(* IEC 61131-3 sources: volt/packages/volt-lsp-iec/test-corpus/lenze-mid/Device/Plc Logic/Application/Library Manager/L_MC4P_RoboticHandling (part 3) *)

(* ---- L_MC4P_KIN_REF_GENERIC.pou ---- *)
FUNCTION_BLOCK L_MC4P_KIN_REF_GENERIC
VAR_OUTPUT
	XACTIVE : BOOL;
END_VAR
VAR
	PAXESGROUP : POINTER TO Axes_Group_KIN;
END_VAR
END_FUNCTION_BLOCK

METHOD GETPARAITF : L_MC4P_IKinParamExtern
END_METHOD

METHOD GETTRAFOITF : L_MC4P_ITrafoExtern
END_METHOD

METHOD LINKEDAXESGROUP_GET : POINTER TO AXES_GROUP_KIN
END_METHOD

METHOD LINKEDAXESGROUP_SET
VAR_INPUT
	LINKEDAXESGROUP : POINTER TO AXES_GROUP_KIN;
END_VAR
END_METHOD

METHOD SETACSAXISTYPE
VAR_OUTPUT
	AEAXES : ARRAY [1..6] OF L_MC4P_AxisType := [L_MC4P_AxisType.linear, L_MC4P_AxisType.linear, L_MC4P_AxisType.linear, L_MC4P_AxisType.rotary, L_MC4P_AxisType.unconnected, L_MC4P_AxisType.unconnected];
END_VAR
END_METHOD

METHOD SETINITIALVALUESOFCONSTANTMCSAXES
VAR_OUTPUT
	ALRMCSPOS : ARRAY [1..6] OF LREAL := [0.0, 0.0, 0.0, 180.0, 0.0, 0.0];
END_VAR
END_METHOD

METHOD SETMCSAXISTYPE
VAR_OUTPUT
	AEAXES : ARRAY [1..6] OF L_MC4P_AxisType := [L_MC4P_AxisType.linear, L_MC4P_AxisType.linear, L_MC4P_AxisType.linear, L_MC4P_AxisType.unconnected, L_MC4P_AxisType.unconnected, L_MC4P_AxisType.rotary];
END_VAR
END_METHOD

METHOD CALCULATEPARAMETER
END_METHOD

METHOD CHECKPARAMETER : BOOL
END_METHOD

METHOD PARAMETERCHANGED
END_METHOD

METHOD CALCBACKWARDTRAFO : WORD
VAR_IN_OUT
	AXESGROUP : AXES_GROUP_KIN;
	ALRPOSFLANGE : ARRAY [1..6] OF LREAL;
	ALRPOSAXES : ARRAY [1..6] OF LREAL;
	AICONFIGURATION : ARRAY [1..6] OF INT;
END_VAR
END_METHOD

METHOD CALCFORWARDTRAFO : WORD
VAR_IN_OUT
	AXESGROUP : AXES_GROUP_KIN;
	ALRPOSFLANGE : ARRAY [1..6] OF LREAL;
	ALRPOSAXES : ARRAY [1..6] OF LREAL;
END_VAR
END_METHOD

METHOD CALCULATECONFIGURATION : WORD
VAR_IN_OUT
	AXESGROUP : AXES_GROUP_KIN;
	ALRPOSFLANGE : ARRAY [1..6] OF LREAL;
	ALRPOSAXES : ARRAY [1..6] OF LREAL;
	AICONFIGURATION : ARRAY [1..6] OF INT;
END_VAR
END_METHOD

(* ---- L_MC4P_KINCOORDPROVIDER.pou ---- *)
FUNCTION_BLOCK L_MC4P_KINCOORDPROVIDER
VAR_INPUT
	ALRACSPOS : ARRAY [1..6] OF LREAL;
	ALRACSVEL : ARRAY [1..6] OF LREAL;
	ALRACSACC : ARRAY [1..6] OF LREAL;
	ALRJCSPOS : ARRAY [1..6] OF LREAL;
	ALRJCSVEL : ARRAY [1..6] OF LREAL;
	ALRJCSACC : ARRAY [1..6] OF LREAL;
	ALRFCSPOS : ARRAY [1..6] OF LREAL;
	ALRFCSVEL : ARRAY [1..6] OF LREAL;
	ALRFCSACC : ARRAY [1..6] OF LREAL;
	ALRMCSPOS : ARRAY [1..6] OF LREAL;
	ALRMCSVEL : ARRAY [1..6] OF LREAL;
	ALRMCSACC : ARRAY [1..6] OF LREAL;
	ALRWCSPOS : ARRAY [1..6] OF LREAL;
	ALRWCSVEL : ARRAY [1..6] OF LREAL;
	ALRWCSACC : ARRAY [1..6] OF LREAL;
	SCFCSFRAME : L_UMTP_RobotFrame;
	SCMCSFRAME : L_UMTP_RobotFrame;
	SCWCSFRAME : L_UMTP_RobotFrame;
END_VAR
VAR_OUTPUT
	UDILOWERSYSTEM : UDINT := 0;
	UDIUPPERSYSTEM : UDINT := 0;
	UDIDIM : UDINT := 0;
	PLRACSPOS : POINTER TO LREAL;
	PLRACSVEL : POINTER TO LREAL;
	PLRACSACC : POINTER TO LREAL;
	PLRJCSPOS : POINTER TO LREAL;
	PLRJCSVEL : POINTER TO LREAL;
	PLRJCSACC : POINTER TO LREAL;
	PLRFCSPOS : POINTER TO LREAL;
	PLRFCSVEL : POINTER TO LREAL;
	PLRFCSACC : POINTER TO LREAL;
	PLRMCSPOS : POINTER TO LREAL;
	PLRMCSVEL : POINTER TO LREAL;
	PLRMCSACC : POINTER TO LREAL;
	PLRWCSPOS : POINTER TO LREAL;
	PLRWCSVEL : POINTER TO LREAL;
	PLRWCSACC : POINTER TO LREAL;
	PFCSFRAME : POINTER TO L_UMTP_RobotFrame;
	PMCSFRAME : POINTER TO L_UMTP_RobotFrame;
	PWCSFRAME : POINTER TO L_UMTP_RobotFrame;
END_VAR
VAR
	ACSACC : POINTER TO LREAL;
	ACSPOS : POINTER TO LREAL;
	ACSVEL : POINTER TO LREAL;
	DIM : UDINT;
	FCSACC : POINTER TO LREAL;
	FCSFRAME : POINTER TO L_UMTP_RobotFrame;
	FCSPOS : POINTER TO LREAL;
	FCSVEL : POINTER TO LREAL;
	JCSACC : POINTER TO LREAL;
	JCSPOS : POINTER TO LREAL;
	JCSVEL : POINTER TO LREAL;
	LOWERSYSTEM : UDINT;
	MCSACC : POINTER TO LREAL;
	MCSFRAME : POINTER TO L_UMTP_RobotFrame;
	MCSPOS : POINTER TO LREAL;
	MCSVEL : POINTER TO LREAL;
	UPPERSYSTEM : UDINT;
	WCSACC : POINTER TO LREAL;
	WCSFRAME : POINTER TO L_UMTP_RobotFrame;
	WCSPOS : POINTER TO LREAL;
	WCSVEL : POINTER TO LREAL;
END_VAR
END_FUNCTION_BLOCK

METHOD EQUALS : BOOL
VAR_INPUT
	ITFPROVIDER : L_MC4P_IKinCoordProvider;
	UDISYSTEM : UDINT;
	XPOS : BOOL;
	XVEL : BOOL;
	XACC : BOOL;
END_VAR
END_METHOD

METHOD FB_INIT : BOOL
VAR_INPUT
	BINITRETAINS : BOOL;
	BINCOPYCODE : BOOL;
END_VAR
END_METHOD

METHOD FB_REINIT : BOOL
END_METHOD

METHOD COPYFRAME
VAR_INPUT
	PSCFRAME : POINTER TO L_UMTP_RobotFrame;
END_VAR
VAR_IN_OUT
	SCFRAME : L_UMTP_RobotFrame;
END_VAR
END_METHOD

METHOD COPYVECTOR
VAR_INPUT
	PLR : POINTER TO LREAL;
END_VAR
VAR_IN_OUT
	ALR : ARRAY [1..6] OF LREAL;
END_VAR
END_METHOD

METHOD CLEAR
END_METHOD

METHOD COPYFROM
VAR_INPUT
	ICOORD : L_MC4P_IKinCoordProvider;
	ELEVEL : INT;
END_VAR
END_METHOD

METHOD SETDIM
VAR_INPUT
	UDIDIM : UDINT;
END_VAR
END_METHOD

METHOD SETLOWERSYSTEM
VAR_INPUT
	UDILOWER : UDINT;
END_VAR
END_METHOD

METHOD SETUPPERSYSTEM
VAR_INPUT
	UDIUPPER : UDINT;
END_VAR
END_METHOD

METHOD THRESHOLD
VAR_INPUT
	LRTHRESHOLD : LREAL;
END_VAR
END_METHOD

(* ---- L_MC4P_KINEMATIKPARAM.pou ---- *)
FUNCTION_BLOCK L_MC4P_KINEMATIKPARAM
VAR_INPUT
	ITFEXTKINPARAM : L_MC4P_IKinParamExtern;
END_VAR
END_FUNCTION_BLOCK

METHOD CALCULATEPARAMETER
END_METHOD

METHOD CHECKPARAMETER : BOOL
END_METHOD

(* ---- L_MC4P_LIMITDYNAMICSAUXAXES.pou ---- *)
FUNCTION_BLOCK L_MC4P_LIMITDYNAMICSAUXAXES EXTENDS L_MC4P_LimitDynamicsAxes
VAR_INPUT
	XENABLE : BOOL;
	ALRMAXAXESVEL : ARRAY [1..6] OF LREAL;
	ALRMAXAXESACC : ARRAY [1..6] OF LREAL;
	ALRMAXAXESJERK : ARRAY [1..6] OF LREAL;
END_VAR
VAR_OUTPUT
	XVALID : BOOL;
	XBUSY : BOOL;
	XERROR : BOOL;
	EERRORID : L_IE1P_Error := L_IE1P_Error.NoError;
END_VAR
END_FUNCTION_BLOCK

(* ---- L_MC4P_LIMITDYNAMICSAXES.pou ---- *)
FUNCTION_BLOCK L_MC4P_LIMITDYNAMICSAXES EXTENDS L_MC4P_Template_AG_KIN
VAR
	XENABLEOLD : BOOL;
	IDX : WORD;
END_VAR
END_FUNCTION_BLOCK

METHOD MAIN
VAR_INPUT
	XENABLE : BOOL;
	ALRMAXAXESVEL : ARRAY [1..6] OF LREAL;
	ALRMAXAXESACC : ARRAY [1..6] OF LREAL;
	ALRMAXAXESJERK : ARRAY [1..6] OF LREAL;
	AXESOFFSET : WORD;
END_VAR
VAR_OUTPUT
	XVALID : BOOL;
	XBUSY : BOOL;
	XERROR : BOOL;
	EERRORID : L_IE1P_Error := L_IE1P_Error.NoError;
END_VAR
VAR_IN_OUT
	AXESGROUP : AXES_GROUP_KIN;
END_VAR
END_METHOD

(* ---- L_MC4P_LIMITDYNAMICSMAINAXES.pou ---- *)
FUNCTION_BLOCK L_MC4P_LIMITDYNAMICSMAINAXES EXTENDS L_MC4P_LimitDynamicsAxes
VAR_INPUT
	XENABLE : BOOL;
	ALRMAXAXESVEL : ARRAY [1..6] OF LREAL;
	ALRMAXAXESACC : ARRAY [1..6] OF LREAL;
	ALRMAXAXESJERK : ARRAY [1..6] OF LREAL;
END_VAR
VAR_OUTPUT
	XVALID : BOOL;
	XBUSY : BOOL;
	XERROR : BOOL;
	EERRORID : L_IE1P_Error := L_IE1P_Error.NoError;
END_VAR
END_FUNCTION_BLOCK

(* ---- L_MC4P_LIMITDYNAMICSREALAXES.pou ---- *)
FUNCTION_BLOCK L_MC4P_LIMITDYNAMICSREALAXES EXTENDS L_MC4P_LimitDynamicsAxes
VAR_INPUT
	XENABLE : BOOL;
	ALRMAXAXESVEL : ARRAY [1..6] OF LREAL;
	ALRMAXAXESACC : ARRAY [1..6] OF LREAL;
	ALRMAXAXESJERK : ARRAY [1..6] OF LREAL;
END_VAR
VAR_OUTPUT
	XVALID : BOOL;
	XBUSY : BOOL;
	XERROR : BOOL;
	EERRORID : L_IE1P_Error := L_IE1P_Error.NoError;
END_VAR
END_FUNCTION_BLOCK

(* ---- L_MC4P_LISTELMINFO.pou ---- *)
FUNCTION_BLOCK L_MC4P_LISTELMINFO
VAR_INPUT
	XENABLE : BOOL;
	UDIELMIDX : UDINT := 1;
END_VAR
VAR_OUTPUT
	XBUSY : BOOL;
	XERROR : BOOL;
	EERRORID : L_IE1P_Error;
	XVALIDELM : BOOL;
	LRVMAX : LREAL;
	LRAMAX : LREAL;
	LRDMAX : LREAL;
	LRJMAX : LREAL;
	ORIGIN_X0 : ARRAY [1..6] OF LREAL;
	ORIGIN_X1 : ARRAY [1..6] OF LREAL;
	ORIGIN_X0_PTP : ARRAY [1..6] OF LREAL;
	ORIGIN_X1_PTP : ARRAY [1..6] OF LREAL;
	X0 : ARRAY [1..6] OF LREAL;
	X1 : ARRAY [1..6] OF LREAL;
	X0_PTP : ARRAY [1..6] OF LREAL;
	X1_PTP : ARRAY [1..6] OF LREAL;
	PPROFILEDATAXYZ : POINTER TO L_MC1P_ProfileData;
	DWMASK : L_MC4P_ModulMask;
END_VAR
VAR_IN_OUT
	AXESGROUP : AXES_GROUP_KIN;
END_VAR
VAR
	_MODEL : L_UBUP_BehaviourModel_LConC;
END_VAR
END_FUNCTION_BLOCK

METHOD CYCLICACTION
VAR_INPUT
	ITFTIMINGCONTROLLER : L_UBUP_ITimingController;
END_VAR
VAR_OUTPUT
	XCOMPLETE : BOOL;
	XABORT : BOOL;
	IERRORID : INT;
END_VAR
END_METHOD

METHOD FINALIZEACTION
VAR_INPUT
	XABORTPROPOSED : BOOL;
	IERRORIDPROPOSED : INT;
END_VAR
VAR_OUTPUT
	XCOMPLETE : BOOL;
	XABORT : BOOL;
	IERRORID : INT;
END_VAR
END_METHOD

METHOD RESETACTION
VAR_OUTPUT
	XCOMPLETE : BOOL;
END_VAR
END_METHOD

METHOD STARTACTION
VAR_OUTPUT
	XCOMPLETE : BOOL;
	IERRORID : INT;
END_VAR
END_METHOD

(* ---- L_MC4P_MFUNCTIONFROMPATHREF.pou ---- *)
FUNCTION_BLOCK L_MC4P_MFUNCTIONFROMPATHREF
VAR_INPUT
	PATHREF : MC_PATH_REF;
	XENABLE : BOOL;
	WMFUNCTION : WORD;
END_VAR
VAR_OUTPUT
	XBUSY : BOOL;
	XACTIVE : BOOL;
	XWAITINGFORMACKNOWLEDGE : BOOL;
	XERROR : BOOL;
	EERRORID : L_IE1P_Error;
	SCPARAMS : L_MC4P_MParams;
END_VAR
VAR
	REQUESTSINFO : DWORD;
	REQUESTSINFO_OLD : DWORD;
	DWRTRIG : DWORD;
	DWFTRIG : DWORD;
	XPATHREFVALID : BOOL;
	XWPATHREFID : __XWORD;
	DWPATHREFSTATUS : DWORD;
	XPATHREFERROR : BOOL;
	PELEMENT : POINTER TO L_MC4P_Parameter_MCMove;
	XIPOACTIVE : BOOL;
	XIPODONE : BOOL;
	XPARAMDIALOG : BOOL := FALSE;
	IVISUMPARAMI0 : INT := 1;
	PALRPARAMSACCESS : POINTER TO ARRAY [1..26] OF LREAL;
	ALRPARAMNAME : ARRAY [1..26] OF WSTRING := ["PA", "PB", "PC", "PD", "PE", "PF", "PG", "PH", "PI", "PJ", "PK", "PL", "PM", "PN", "PO", "PP", "PQ", "PR", "PS", "PT", "PU", "PV", "PW", "PX", "PY", "PZ"];
END_VAR
END_FUNCTION_BLOCK

METHOD CALL_ALLOCPOINTADR
END_METHOD

METHOD CALL_ERRORHANDLER
VAR_IN_OUT
	PATHREF : MC_PATH_REF;
END_VAR
END_METHOD

METHOD CALL_OUTPUT
END_METHOD

METHOD CALL_PATHREFINFO
END_METHOD

METHOD CALL_REQUESTS_EXT
END_METHOD

METHOD CALL_RESETOUTPUT
END_METHOD

METHOD CALL_STATEMACHINE
VAR_IN_OUT
	PATHREF : MC_PATH_REF;
END_VAR
END_METHOD

METHOD FB_INIT : BOOL
VAR_INPUT
	BINITRETAINS : BOOL;
	BINCOPYCODE : BOOL;
END_VAR
END_METHOD

(* ---- L_MC4P_MOVECIRCULARABSOLUTE_INTERNAL.pou ---- *)
FUNCTION_BLOCK L_MC4P_MOVECIRCULARABSOLUTE_INTERNAL EXTENDS L_MC4P_MoveContPath
VAR_INPUT
	EXECUTE : BOOL;
	CIRCMODE : L_MC4P_CircMode;
	AUXPOINT : ARRAY [1..12] OF LREAL;
	ENDPOINT : ARRAY [1..12] OF LREAL;
	PATHCHOICE : MC_CIRC_PATHCHOICE;
	VELOCITY : LREAL;
	ACCELERATION : LREAL;
	DECELERATION : LREAL;
	JERK : LREAL;
	COORDSYSTEM : L_MC4P_CoordSystem;
	BUFFERMODE : MC_BUFFER_MODE;
	TRANSITIONMODE : MC_TRANSITION_MODE;
	TRANSITIONPARAMETER : ARRAY [1..12] OF LREAL := [12(0)];
	AEAUXMODE : ARRAY [1..6] OF L_MC4P_AuxMode;
	ORIENTATIONMODE : L_MC4P_Orientation_Mode := L_MC4P_Orientation_Mode.ShortestSpacialWay;
	DIRECTION : ARRAY [4..6] OF MC_DIRECTION := [3(MC_DIRECTION.mcShortestWay)];
END_VAR
VAR_OUTPUT
	DONE : BOOL;
	BUSY : BOOL;
	ACTIVE : BOOL;
	COMMANDABORTED : BOOL;
	ERROR : BOOL;
	ERRORID : L_IE1P_Error;
END_VAR
VAR
	CLASSID : DINT;
END_VAR
END_FUNCTION_BLOCK

METHOD HOMINGREQUIRED : BOOL
END_METHOD

METHOD MAIN
VAR_IN_OUT
	AXESGROUP : AXES_GROUP_KIN;
	FBBASE : L_MC4P_Template_AG_KIN;
END_VAR
END_METHOD

METHOD PARAMETERFREEZE
VAR_IN_OUT
	AXESGROUP : AXES_GROUP_KIN;
	FBBASE : L_MC4P_Template_AG_KIN;
	COORDSYSTEM : L_MC4P_CoordSystem;
	BUFFERMODE : MC_BUFFER_MODE;
	TRANSITIONMODE : MC_TRANSITION_MODE;
	TRANSITIONPARAMETER : ARRAY [1..12] OF LREAL;
END_VAR
END_METHOD

METHOD SETERRORINPUTLIMITATIONVIOLATION
VAR_IN_OUT
	FBBASE : L_MC4P_Template_AG_KIN;
END_VAR
END_METHOD

METHOD SETPATHELEMENT
VAR_IN_OUT
	AXESGROUP : AXES_GROUP_KIN;
	FBBASE : L_MC4P_Template_AG_KIN;
	ALRSTARTPOS : ARRAY [1..12] OF LREAL;
	ALRSUPERPOSPOSATSTART : ARRAY [1..3] OF LREAL;
END_VAR
END_METHOD

(* ---- L_MC4P_MOVECIRCULARRELATIVE_INTERNAL.pou ---- *)
FUNCTION_BLOCK L_MC4P_MOVECIRCULARRELATIVE_INTERNAL EXTENDS L_MC4P_MoveContPath
VAR_INPUT
	EXECUTE : BOOL;
	CIRCMODE : L_MC4P_CircMode;
	AUXPOINT : ARRAY [1..12] OF LREAL;
	ENDPOINT : ARRAY [1..12] OF LREAL;
	PATHCHOICE : MC_CIRC_PATHCHOICE;
	VELOCITY : LREAL;
	ACCELERATION : LREAL;
	DECELERATION : LREAL;
	JERK : LREAL;
	COORDSYSTEM : L_MC4P_CoordSystem;
	BUFFERMODE : MC_BUFFER_MODE;
	TRANSITIONMODE : MC_TRANSITION_MODE;
	TRANSITIONPARAMETER : ARRAY [1..12] OF LREAL := [12(0)];
	AEAUXMODE : ARRAY [1..6] OF L_MC4P_AuxMode;
	ORIENTATIONMODE : L_MC4P_Orientation_Mode := L_MC4P_Orientation_Mode.ShortestSpacialWay;
	DIRECTION : ARRAY [4..6] OF MC_DIRECTION := [3(MC_DIRECTION.mcShortestWay)];
END_VAR
VAR_OUTPUT
	DONE : BOOL;
	BUSY : BOOL;
	ACTIVE : BOOL;
	COMMANDABORTED : BOOL;
	ERROR : BOOL;
	ERRORID : L_IE1P_Error;
END_VAR
VAR
	CLASSID : DINT;
END_VAR
END_FUNCTION_BLOCK

METHOD HOMINGREQUIRED : BOOL
END_METHOD

METHOD MAIN
VAR_IN_OUT
	AXESGROUP : AXES_GROUP_KIN;
	FBBASE : L_MC4P_Template_AG_KIN;
END_VAR
END_METHOD

METHOD PARAMETERFREEZE
VAR_IN_OUT
	AXESGROUP : AXES_GROUP_KIN;
	FBBASE : L_MC4P_Template_AG_KIN;
	COORDSYSTEM : L_MC4P_CoordSystem;
	BUFFERMODE : MC_BUFFER_MODE;
	TRANSITIONMODE : MC_TRANSITION_MODE;
	TRANSITIONPARAMETER : ARRAY [1..12] OF LREAL;
END_VAR
END_METHOD

METHOD SETERRORINPUTLIMITATIONVIOLATION
VAR_IN_OUT
	FBBASE : L_MC4P_Template_AG_KIN;
END_VAR
END_METHOD

METHOD SETPATHELEMENT
VAR_IN_OUT
	AXESGROUP : AXES_GROUP_KIN;
	FBBASE : L_MC4P_Template_AG_KIN;
	ALRSTARTPOS : ARRAY [1..12] OF LREAL;
	ALRSUPERPOSPOSATSTART : ARRAY [1..3] OF LREAL;
END_VAR
END_METHOD

(* ---- L_MC4P_MOVECONTPATH.pou ---- *)
FUNCTION_BLOCK L_MC4P_MOVECONTPATH EXTENDS L_UBUP_PoolInstance
VAR_INPUT
	LRCONVEYORPOSEXTRAPOL : LREAL;
	XDONTCALCPROFILEMOVEPATH : BOOL;
	ITFPATHELMDELETE : L_MC4P_IPathElmDelete;
	ITFTOOLINFO : L_MC4P_IToolInfo;
	ESRCOFCMD : L_MC4P_SourceOfMotionCommand := L_MC4P_SourceOfMotionCommand.ContPathPrepare;
END_VAR
VAR
	CALCSTOPPROFILES : L_MC4P_CalcStopProfiles;
	XMOVEREL : BOOL;
	XDONTCHECKTARGETPOSSWLIMITS : BOOL;
	XDONE_INTERN : BOOL;
	XBUSY_INTERN : BOOL;
	XACTIVE_INTERN : BOOL;
	XCOMMANDABORTED_INTERN : BOOL;
	XERROR_INTERN : BOOL;
	EERRORID_INTERN : L_IE1P_Error;
	INPUT_PARAMETER : L_MC4P_Parameter_MCMove;
	COORDTRAFOPCSFORTMPUSE : L_MC4P_CoordTrafo;
	SCPATHELEMENT : L_MC4P_PathElement;
	DIFUNID : DINT := -1;
	EXECUTEOLD : BOOL;
	WSTEP : L_MC4P_MoveContStates := L_MC4P_MoveContStates.Initial;
	WSTEPOLD : L_MC4P_MoveContStates := L_MC4P_MoveContStates.Initial;
	ALRSTARTPOS : ARRAY [1..12] OF LREAL;
	ALRPOSITIONATEXECUTE : ARRAY [1..18] OF LREAL;
	BSTATEMACHINE : BOOL;
	IPO_DONE : BOOL;
	WMASTEROFIPO : WORD;
	ERROROLD : BOOL;
	XRESETOUTPUT : BOOL := FALSE;
	SINSTANCESTR : STRING;
	ISPLINEPOINTPASSED_INTERN : INT;
	XINITABORTING : BOOL;
	PTRACKINGPARAM : POINTER TO L_MC4P_PCSTrackParam;
	PSCHANDSHAKE : POINTER TO L_MC4P_TrackingHandshake;
	XWINSTANCE : __XWORD;
	XMOVEPATHEXECUTE : BOOL;
	PSCPARMOVEPATH : POINTER TO L_MC4P_Parameter_MCMove;
	XTIMEIPOACTIVE : BOOL;
	LRCIRCANGLEEXTENDED : LREAL;
	CLASSID : DINT;
	TARGETREACHED : BOOL;
END_VAR
END_FUNCTION_BLOCK

METHOD CALCTARGETPOSITION : L_IE1P_Error
VAR_INPUT
	COORDSYSTEM : L_MC4P_CoordSystem;
	XCALCACSPOS : BOOL;
END_VAR
VAR_IN_OUT
	AXESGROUP : AXES_GROUP_KIN;
	FBBASE : L_MC4P_Template_AG_KIN;
	ALRSTARTPOS : ARRAY [1..12] OF LREAL;
	ALRPOS : ARRAY [1..12] OF LREAL;
	ALRTARGETPOS : ARRAY [1..12] OF LREAL;
	ALRTARGETPOSAUX : ARRAY [1..6] OF LREAL;
	SCTRAFOINFO : L_MC4P_TrafoInfo;
END_VAR
END_METHOD

METHOD CHECKIPOVALUES : BOOL
VAR_INPUT
	LRVELTOCHECK : LREAL;
	LRACCTOCHECK : LREAL;
	LRMAXVEL : LREAL;
	LRMAXACCDEC : LREAL;
	LRMAXJERK : LREAL;
END_VAR
VAR_IN_OUT
	AXESGROUP : AXES_GROUP_KIN;
END_VAR
END_METHOD

METHOD FB_INIT : BOOL
VAR_INPUT
	BINITRETAINS : BOOL;
	BINCOPYCODE : BOOL;
END_VAR
END_METHOD

METHOD GETPROFILETIME : LREAL
VAR_IN_OUT
	AXESGROUP : AXES_GROUP_KIN;
END_VAR
END_METHOD

METHOD GETREMAININGSEGMENTLENGTH : LREAL
VAR_IN_OUT
	AXESGROUP : AXES_GROUP_KIN;
END_VAR
END_METHOD

METHOD GETREMAININGSEGMENTTIME : BOOL
VAR_INPUT
	LRDISTANCETOTARGET : LREAL;
END_VAR
VAR_OUTPUT
	LRREMAININGTIME : LREAL;
END_VAR
VAR_IN_OUT
	AXESGROUP : AXES_GROUP_KIN;
END_VAR
END_METHOD

METHOD HOMINGREQUIRED : BOOL
END_METHOD

METHOD ISPTP : BOOL
END_METHOD

METHOD LIMITCP2AXESGROUPLIMITS : L_IE1P_Error
VAR_INPUT
	EPATHVELERRORID : L_IE1P_Error;
	EPATHACCERRORID : L_IE1P_Error;
	EPATHDECERRORID : L_IE1P_Error;
	EPATHJERKERRORID : L_IE1P_Error;
	EROTVELERRORID : L_IE1P_Error;
	EROTACCERRORID : L_IE1P_Error;
	EROTJERKERRORID : L_IE1P_Error;
	ETRANSPARAERRORID : L_IE1P_Error;
	ETRANSMODEERRORID : L_IE1P_Error;
END_VAR
VAR_IN_OUT
	AXESGROUP : AXES_GROUP_KIN;
	FBBASE : L_MC4P_Template_AG_KIN;
	AEAUXMODE : ARRAY [1..6] OF L_MC4P_AuxMode;
END_VAR
END_METHOD

METHOD PARAMETERFREEZE
VAR_IN_OUT
	AXESGROUP : AXES_GROUP_KIN;
	FBBASE : L_MC4P_Template_AG_KIN;
	COORDSYSTEM : L_MC4P_CoordSystem;
	BUFFERMODE : MC_BUFFER_MODE;
	TRANSITIONMODE : MC_TRANSITION_MODE;
	TRANSITIONPARAMETER : ARRAY [1..12] OF LREAL;
END_VAR
END_METHOD

METHOD SETERRORINPUTLIMITATIONVIOLATION
VAR_IN_OUT
	FBBASE : L_MC4P_Template_AG_KIN;
END_VAR
END_METHOD

METHOD SETPATHELEMENT_CARTESIAN
VAR_IN_OUT
	AXESGROUP : AXES_GROUP_KIN;
	FBBASE : L_MC4P_Template_AG_KIN;
	ALRSTARTPOS : ARRAY [1..12] OF LREAL;
	ALRSUPERPOSPOSATSTART : ARRAY [1..3] OF LREAL;
	AEAUXMODE : ARRAY [1..6] OF L_MC4P_AuxMode;
END_VAR
END_METHOD

METHOD SETIPO_DONE
VAR_INPUT
	IPO_DONE : BOOL;
END_VAR
END_METHOD

METHOD SETINSTANCESTRING
VAR_INPUT
	SINSTANCESTR_FATHER : STRING;
END_VAR
END_METHOD

METHOD SETMASTEROFIPO
VAR_INPUT
	WSETMASTEROFIPO : WORD;
END_VAR
END_METHOD

METHOD SETMOVECONTSTATE
VAR_INPUT
	WNEWSTEP : L_MC4P_MoveContStates;
END_VAR
END_METHOD

METHOD SETTIMEIPOACTIVEFLAG
VAR_INPUT
	XACTIVE : BOOL;
END_VAR
END_METHOD

METHOD GET_EERRORID : L_IE1P_Error
END_METHOD

METHOD GET_XACTIVE : BOOL
END_METHOD

METHOD GET_XBUSY : BOOL
END_METHOD

METHOD GET_XCOMMANDABORTED : BOOL
END_METHOD

METHOD GET_XDONE : BOOL
END_METHOD

METHOD GET_XINITIAL : BOOL
END_METHOD

METHOD FREE : BOOL
END_METHOD

METHOD REQUESTINTERFACE : BOOL
VAR_INPUT
	ID : DINT;
	PITFUNKNOWN : POINTER TO L_UBUP_IUnknown;
END_VAR
END_METHOD

METHOD CALCCIRCULARBORDERMODE : L_IE1P_Error
VAR_IN_OUT
	AXESGROUP : AXES_GROUP_KIN;
	FBBASE : L_MC4P_Template_AG_KIN;
END_VAR
END_METHOD

METHOD CALCCIRCULARCENTERMODE : L_IE1P_Error
VAR_INPUT
	ALRSTARTPOS : ARRAY [1..12] OF LREAL;
END_VAR
VAR_IN_OUT
	AXESGROUP : AXES_GROUP_KIN;
	FBBASE : L_MC4P_Template_AG_KIN;
END_VAR
END_METHOD

METHOD CALCCIRCULARRADIUSMODE : L_IE1P_Error
VAR_INPUT
	ALRSTARTPOS : ARRAY [1..12] OF LREAL;
END_VAR
VAR_IN_OUT
	AXESGROUP : AXES_GROUP_KIN;
	FBBASE : L_MC4P_Template_AG_KIN;
END_VAR
END_METHOD

METHOD SETPATHELEMENT_CIRCULAR
VAR_IN_OUT
	AXESGROUP : AXES_GROUP_KIN;
	FBBASE : L_MC4P_Template_AG_KIN;
	ALRSTARTPOS : ARRAY [1..12] OF LREAL;
	ALRSUPERPOSPOSATSTART : ARRAY [1..3] OF LREAL;
	AEAUXMODE : ARRAY [1..6] OF L_MC4P_AuxMode;
END_VAR
END_METHOD

METHOD SETPATHELEMENT_DIRECT
VAR_IN_OUT
	AXESGROUP : AXES_GROUP_KIN;
	FBBASE : L_MC4P_Template_AG_KIN;
	ALRSTARTPOS : ARRAY [1..12] OF LREAL;
	ALRSUPERPOSPOSATSTART : ARRAY [1..3] OF LREAL;
	AEAUXMODE : ARRAY [1..6] OF L_MC4P_AuxMode;
END_VAR
END_METHOD

METHOD CALCELLIPSE180DEG : L_IE1P_Error
VAR_INPUT
	ALRSTARTPOS : ARRAY [1..12] OF LREAL;
END_VAR
END_METHOD

METHOD CALCELLIPSE90DEG : L_IE1P_Error
VAR_INPUT
	ALRSTARTPOS : ARRAY [1..12] OF LREAL;
END_VAR
END_METHOD

METHOD CALCELLIPSECENTERMODE : L_IE1P_Error
VAR_INPUT
	ALRSTARTPOS : ARRAY [1..12] OF LREAL;
END_VAR
END_METHOD

METHOD SETPATHELEMENT_ELLIPTICAL
VAR_IN_OUT
	AXESGROUP : AXES_GROUP_KIN;
	FBBASE : L_MC4P_Template_AG_KIN;
	ALRSTARTPOS : ARRAY [1..12] OF LREAL;
	ALRSUPERPOSPOSATSTART : ARRAY [1..3] OF LREAL;
	AEAUXMODE : ARRAY [1..6] OF L_MC4P_AuxMode;
END_VAR
END_METHOD

METHOD SETPATHELEMENT_ELLIPTICALPNP
VAR_IN_OUT
	AXESGROUP : AXES_GROUP_KIN;
	FBBASE : L_MC4P_Template_AG_KIN;
	ALRSTARTPOS : ARRAY [1..12] OF LREAL;
	ALRSUPERPOSPOSATSTART : ARRAY [1..3] OF LREAL;
	AEAUXMODE : ARRAY [1..6] OF L_MC4P_AuxMode;
END_VAR
END_METHOD

METHOD SETPATHELEMENT_LINEAR
VAR_IN_OUT
	AXESGROUP : AXES_GROUP_KIN;
	FBBASE : L_MC4P_Template_AG_KIN;
	ALRSTARTPOS : ARRAY [1..12] OF LREAL;
	ALRSUPERPOSPOSATSTART : ARRAY [1..3] OF LREAL;
	AEAUXMODE : ARRAY [1..6] OF L_MC4P_AuxMode;
END_VAR
END_METHOD

METHOD MOVEMCMOVEPATH
VAR_IN_OUT
	XPAUSE : BOOL;
	AXESGROUP : AXES_GROUP_KIN;
	FBBASE : L_MC4P_Template_AG_KIN;
	SCPARMOVEPATH : L_MC4P_Parameter_MCMove;
	XDONE : BOOL;
	XBUSY : BOOL;
	XACTIVE : BOOL;
	XCOMMANDABORTED : BOOL;
	XERROR : BOOL;
	EERRORID : L_IE1P_Error;
END_VAR
END_METHOD

METHOD MOVEPATHDECODECIRCULAR
VAR_IN_OUT
	AXESGROUP : AXES_GROUP_KIN;
	FBBASE : L_MC4P_Template_AG_KIN;
	ALRSTARTPOS : ARRAY [1..12] OF LREAL;
END_VAR
END_METHOD

METHOD MOVEPATHINPUT
VAR_IN_OUT
	SCPARMOVEPATH : L_MC4P_Parameter_MCMove;
END_VAR
END_METHOD

METHOD PARAMETERFREEZE_MOVEPATH
VAR_IN_OUT
	AXESGROUP : AXES_GROUP_KIN;
	FBBASE : L_MC4P_Template_AG_KIN;
END_VAR
END_METHOD

METHOD SETPATHELEMENT
VAR_IN_OUT
	AXESGROUP : AXES_GROUP_KIN;
	FBBASE : L_MC4P_Template_AG_KIN;
	ALRSTARTPOS : ARRAY [1..12] OF LREAL;
	ALRSUPERPOSPOSATSTART : ARRAY [1..3] OF LREAL;
END_VAR
END_METHOD

METHOD CHECKPOINTS : L_IE1P_Error
VAR_IN_OUT
	ALRSTARTPOS : ARRAY [1..12] OF LREAL;
END_VAR
END_METHOD

METHOD PRECALCPOINTS : L_IE1P_Error
VAR_IN_OUT
	ALRSTARTPOS : ARRAY [1..12] OF LREAL;
	AXESGROUP : AXES_GROUP_KIN;
	FBBASE : L_MC4P_Template_AG_KIN;
END_VAR
END_METHOD

METHOD SETPATHELEMENT_SPLINE
VAR_IN_OUT
	AXESGROUP : AXES_GROUP_KIN;
	FBBASE : L_MC4P_Template_AG_KIN;
	ALRSTARTPOS : ARRAY [1..12] OF LREAL;
	ALRSUPERPOSPOSATSTART : ARRAY [1..3] OF LREAL;
	AEAUXMODE : ARRAY [1..6] OF L_MC4P_AuxMode;
END_VAR
END_METHOD

METHOD SETPATHELEMENT_SPLINEPNP
VAR_IN_OUT
	AXESGROUP : AXES_GROUP_KIN;
	FBBASE : L_MC4P_Template_AG_KIN;
	ALRSTARTPOS : ARRAY [1..12] OF LREAL;
	ALRSUPERPOSPOSATSTART : ARRAY [1..3] OF LREAL;
	AEAUXMODE : ARRAY [1..6] OF L_MC4P_AuxMode;
END_VAR
END_METHOD

METHOD SETSPLINEPOINTPASSED
VAR_INPUT
	UIPOINTPASSED : UINT;
END_VAR
END_METHOD

METHOD MOVECONTPATH
VAR_IN_OUT
	AXESGROUP : AXES_GROUP_KIN;
	FBBASE : L_MC4P_Template_AG_KIN;
	EXECUTE : BOOL;
	COORDSYSTEM : L_MC4P_CoordSystem;
	AEAUXMODE : ARRAY [1..6] OF L_MC4P_AuxMode;
	BUFFERMODE : MC_BUFFER_MODE;
	TRANSITIONMODE : MC_TRANSITION_MODE;
	TRANSITIONPARAMETER : ARRAY [1..12] OF LREAL;
END_VAR
END_METHOD

METHOD MOVECONTSTATES_ABORTING
VAR_IN_OUT
	AXESGROUP : AXES_GROUP_KIN;
	FBBASE : L_MC4P_Template_AG_KIN;
	EXECUTE : BOOL;
	COORDSYSTEM : L_MC4P_CoordSystem;
	AEAUXMODE : ARRAY [1..6] OF L_MC4P_AuxMode;
	BUFFERMODE : MC_BUFFER_MODE;
	TRANSITIONMODE : MC_TRANSITION_MODE;
	TRANSITIONPARAMETER : ARRAY [1..12] OF LREAL;
END_VAR
END_METHOD

METHOD MOVECONTSTATES_CALCPATH
VAR_IN_OUT
	AXESGROUP : AXES_GROUP_KIN;
	FBBASE : L_MC4P_Template_AG_KIN;
	EXECUTE : BOOL;
	COORDSYSTEM : L_MC4P_CoordSystem;
	AEAUXMODE : ARRAY [1..6] OF L_MC4P_AuxMode;
	BUFFERMODE : MC_BUFFER_MODE;
	TRANSITIONMODE : MC_TRANSITION_MODE;
	TRANSITIONPARAMETER : ARRAY [1..12] OF LREAL;
END_VAR
END_METHOD

METHOD MOVECONTSTATES_ERRORSTATE
VAR_IN_OUT
	AXESGROUP : AXES_GROUP_KIN;
	FBBASE : L_MC4P_Template_AG_KIN;
	EXECUTE : BOOL;
	COORDSYSTEM : L_MC4P_CoordSystem;
	AEAUXMODE : ARRAY [1..6] OF L_MC4P_AuxMode;
	BUFFERMODE : MC_BUFFER_MODE;
	TRANSITIONMODE : MC_TRANSITION_MODE;
	TRANSITIONPARAMETER : ARRAY [1..12] OF LREAL;
END_VAR
END_METHOD

METHOD MOVECONTSTATES_IPO_ACTIVE
VAR_IN_OUT
	AXESGROUP : AXES_GROUP_KIN;
	FBBASE : L_MC4P_Template_AG_KIN;
	EXECUTE : BOOL;
	COORDSYSTEM : L_MC4P_CoordSystem;
	AEAUXMODE : ARRAY [1..6] OF L_MC4P_AuxMode;
	BUFFERMODE : MC_BUFFER_MODE;
	TRANSITIONMODE : MC_TRANSITION_MODE;
	TRANSITIONPARAMETER : ARRAY [1..12] OF LREAL;
END_VAR
END_METHOD

METHOD MOVECONTSTATES_IPO_STANDBY
VAR_IN_OUT
	AXESGROUP : AXES_GROUP_KIN;
	FBBASE : L_MC4P_Template_AG_KIN;
	EXECUTE : BOOL;
	COORDSYSTEM : L_MC4P_CoordSystem;
	AEAUXMODE : ARRAY [1..6] OF L_MC4P_AuxMode;
	BUFFERMODE : MC_BUFFER_MODE;
	TRANSITIONMODE : MC_TRANSITION_MODE;
	TRANSITIONPARAMETER : ARRAY [1..12] OF LREAL;
END_VAR
END_METHOD

METHOD MOVECONTSTATES_INITIAL
VAR_IN_OUT
	AXESGROUP : AXES_GROUP_KIN;
	FBBASE : L_MC4P_Template_AG_KIN;
	EXECUTE : BOOL;
	COORDSYSTEM : L_MC4P_CoordSystem;
	AEAUXMODE : ARRAY [1..6] OF L_MC4P_AuxMode;
	BUFFERMODE : MC_BUFFER_MODE;
	TRANSITIONMODE : MC_TRANSITION_MODE;
	TRANSITIONPARAMETER : ARRAY [1..12] OF LREAL;
END_VAR
END_METHOD

METHOD MOVECONTSTATES_READPARAM_STANDBY
VAR_IN_OUT
	AXESGROUP : AXES_GROUP_KIN;
	FBBASE : L_MC4P_Template_AG_KIN;
	EXECUTE : BOOL;
	COORDSYSTEM : L_MC4P_CoordSystem;
	AEAUXMODE : ARRAY [1..6] OF L_MC4P_AuxMode;
	BUFFERMODE : MC_BUFFER_MODE;
	TRANSITIONMODE : MC_TRANSITION_MODE;
	TRANSITIONPARAMETER : ARRAY [1..12] OF LREAL;
END_VAR
END_METHOD

METHOD MOVECONTSTATES_READ_INPUTS
VAR_IN_OUT
	AXESGROUP : AXES_GROUP_KIN;
	FBBASE : L_MC4P_Template_AG_KIN;
	EXECUTE : BOOL;
	COORDSYSTEM : L_MC4P_CoordSystem;
	AEAUXMODE : ARRAY [1..6] OF L_MC4P_AuxMode;
	BUFFERMODE : MC_BUFFER_MODE;
	TRANSITIONMODE : MC_TRANSITION_MODE;
	TRANSITIONPARAMETER : ARRAY [1..12] OF LREAL;
END_VAR
END_METHOD

METHOD SETPATHELEMENT_WAITTIME
VAR_IN_OUT
	AXESGROUP : AXES_GROUP_KIN;
	FBBASE : L_MC4P_Template_AG_KIN;
	ALRSTARTPOS : ARRAY [1..12] OF LREAL;
	ALRSUPERPOSPOSATSTART : ARRAY [1..3] OF LREAL;
	LRWAITTIME : LREAL;
	EERRORID : L_IE1P_Error;
END_VAR
END_METHOD

(* ---- L_MC4P_MOVEDIRECTABSOLUTE_INTERNAL.pou ---- *)
FUNCTION_BLOCK L_MC4P_MOVEDIRECTABSOLUTE_INTERNAL EXTENDS L_MC4P_MoveContPath
VAR_INPUT
	EXECUTE : BOOL;
	POSITION : ARRAY [1..12] OF LREAL;
	COORDSYSTEM : L_MC4P_CoordSystem;
	BUFFERMODE : MC_BUFFER_MODE;
	TRANSITIONMODE : MC_TRANSITION_MODE;
	TRANSITIONPARAMETER : ARRAY [1..12] OF LREAL := [12(0)];
	AITARGETCONFIGURATION : ARRAY [1..6] OF INT;
	DIRECTION : ARRAY [1..6] OF MC_DIRECTION := [6(MC_DIRECTION.mcShortestWay)];
END_VAR
VAR_OUTPUT
	DONE : BOOL;
	BUSY : BOOL;
	ACTIVE : BOOL;
	COMMANDABORTED : BOOL;
	ERROR : BOOL;
	ERRORID : L_IE1P_Error;
END_VAR
VAR
	AEAUXMODE : ARRAY [1..6] OF L_MC4P_AuxMode := [6(L_MC4P_AuxMode.Inactive)];
	CLASSID : DINT;
END_VAR
END_FUNCTION_BLOCK

METHOD HOMINGREQUIRED : BOOL
END_METHOD

METHOD ISPTP : BOOL
END_METHOD

METHOD MAIN
VAR_IN_OUT
	AXESGROUP : AXES_GROUP_KIN;
	FBBASE : L_MC4P_Template_AG_KIN;
END_VAR
END_METHOD

METHOD PARAMETERFREEZE
VAR_IN_OUT
	AXESGROUP : AXES_GROUP_KIN;
	FBBASE : L_MC4P_Template_AG_KIN;
	COORDSYSTEM : L_MC4P_CoordSystem;
	BUFFERMODE : MC_BUFFER_MODE;
	TRANSITIONMODE : MC_TRANSITION_MODE;
	TRANSITIONPARAMETER : ARRAY [1..12] OF LREAL;
END_VAR
END_METHOD

METHOD SETERRORINPUTLIMITATIONVIOLATION
VAR_IN_OUT
	FBBASE : L_MC4P_Template_AG_KIN;
END_VAR
END_METHOD

METHOD SETPATHELEMENT
VAR_IN_OUT
	AXESGROUP : AXES_GROUP_KIN;
	FBBASE : L_MC4P_Template_AG_KIN;
	ALRSTARTPOS : ARRAY [1..12] OF LREAL;
	ALRSUPERPOSPOSATSTART : ARRAY [1..3] OF LREAL;
END_VAR
END_METHOD

(* ---- L_MC4P_MOVEDIRECTRELATIVE_INTERNAL.pou ---- *)
FUNCTION_BLOCK L_MC4P_MOVEDIRECTRELATIVE_INTERNAL EXTENDS L_MC4P_MoveContPath
VAR_INPUT
	EXECUTE : BOOL;
	DISTANCE : ARRAY [1..12] OF LREAL;
	COORDSYSTEM : L_MC4P_CoordSystem;
	BUFFERMODE : MC_BUFFER_MODE;
	TRANSITIONMODE : MC_TRANSITION_MODE;
	TRANSITIONPARAMETER : ARRAY [1..12] OF LREAL := [12(0)];
	AITARGETCONFIGURATION : ARRAY [1..6] OF INT;
	DIRECTION : ARRAY [1..6] OF MC_DIRECTION := [6(MC_DIRECTION.mcShortestWay)];
END_VAR
VAR_OUTPUT
	DONE : BOOL;
	BUSY : BOOL;
	ACTIVE : BOOL;
	COMMANDABORTED : BOOL;
	ERROR : BOOL;
	ERRORID : L_IE1P_Error;
END_VAR
VAR
	AEAUXMODE : ARRAY [1..6] OF L_MC4P_AuxMode := [6(L_MC4P_AuxMode.Inactive)];
	CLASSID : DINT;
END_VAR
END_FUNCTION_BLOCK

METHOD HOMINGREQUIRED : BOOL
END_METHOD

METHOD ISPTP : BOOL
END_METHOD

METHOD MAIN
VAR_IN_OUT
	AXESGROUP : AXES_GROUP_KIN;
	FBBASE : L_MC4P_Template_AG_KIN;
END_VAR
END_METHOD

METHOD PARAMETERFREEZE
VAR_IN_OUT
	AXESGROUP : AXES_GROUP_KIN;
	FBBASE : L_MC4P_Template_AG_KIN;
	COORDSYSTEM : L_MC4P_CoordSystem;
	BUFFERMODE : MC_BUFFER_MODE;
	TRANSITIONMODE : MC_TRANSITION_MODE;
	TRANSITIONPARAMETER : ARRAY [1..12] OF LREAL;
END_VAR
END_METHOD

METHOD SETERRORINPUTLIMITATIONVIOLATION
VAR_IN_OUT
	FBBASE : L_MC4P_Template_AG_KIN;
END_VAR
END_METHOD

METHOD SETPATHELEMENT
VAR_IN_OUT
	AXESGROUP : AXES_GROUP_KIN;
	FBBASE : L_MC4P_Template_AG_KIN;
	ALRSTARTPOS : ARRAY [1..12] OF LREAL;
	ALRSUPERPOSPOSATSTART : ARRAY [1..3] OF LREAL;
END_VAR
END_METHOD

(* ---- L_MC4P_MOVEELLIPTICALABSOLUTE.pou ---- *)
FUNCTION_BLOCK L_MC4P_MOVEELLIPTICALABSOLUTE EXTENDS L_MC4P_Template_MoveLicence
VAR_INPUT
	XEXECUTE : BOOL;
	ALRAUXPOINT : ARRAY [1..12] OF LREAL;
	ALRENDPOINT : ARRAY [1..12] OF LREAL;
	LRSEMIMAJORAXIS : LREAL;
	LRSEMIMINORAXIS : LREAL;
	EPATHCHOICE : MC_CIRC_PATHCHOICE;
	LRVELOCITY : LREAL;
	LRACCELERATION : LREAL;
	LRDECELERATION : LREAL;
	LRJERK : LREAL;
	ECOORDSYSTEM : L_MC4P_CoordSystem;
	EBUFFERMODE : MC_BUFFER_MODE;
	ETRANSITIONMODE : MC_TRANSITION_MODE;
	ALRTRANSITIONPARAMETER : ARRAY [1..12] OF LREAL := [12(0)];
	AEAUXMODE : ARRAY [1..6] OF L_MC4P_AuxMode;
	EORIENTATIONMODE : L_MC4P_Orientation_Mode := L_MC4P_Orientation_Mode.ShortestSpacialWay;
	AEDIRECTION : ARRAY [4..6] OF MC_DIRECTION := [3(MC_DIRECTION.mcShortestWay)];
END_VAR
VAR_OUTPUT
	XDONE : BOOL;
	XBUSY : BOOL;
	XACTIVE : BOOL;
	XCOMMANDABORTED : BOOL;
	XERROR : BOOL;
	EERRORID : L_IE1P_Error;
END_VAR
VAR
	MOVEELLIPTICAL : L_MC4P_MoveEllipticalAbsolute_Internal;
	PMOVE : POINTER TO L_MC4P_MoveContPath;
	SETELLIPTICALTARGETTOLERANCE : LREAL;
END_VAR
END_FUNCTION_BLOCK

(* ---- L_MC4P_MOVEELLIPTICALABSOLUTE_INTERNAL.pou ---- *)
FUNCTION_BLOCK L_MC4P_MOVEELLIPTICALABSOLUTE_INTERNAL EXTENDS L_MC4P_MoveContPath
VAR_INPUT
	XEXECUTE : BOOL;
	ALRAUXPOINT : ARRAY [1..12] OF LREAL;
	ALRENDPOINT : ARRAY [1..12] OF LREAL;
	LRSEMIMAJORAXIS : LREAL;
	LRSEMIMINORAXIS : LREAL;
	EPATHCHOICE : MC_CIRC_PATHCHOICE;
	LRVELOCITY : LREAL;
	LRACCELERATION : LREAL;
	LRDECELERATION : LREAL;
	LRJERK : LREAL;
	ECOORDSYSTEM : L_MC4P_CoordSystem;
	EBUFFERMODE : MC_BUFFER_MODE;
	ETRANSITIONMODE : MC_TRANSITION_MODE;
	ALRTRANSITIONPARAMETER : ARRAY [1..12] OF LREAL := [12(0)];
	AEAUXMODE : ARRAY [1..6] OF L_MC4P_AuxMode;
	EORIENTATIONMODE : L_MC4P_Orientation_Mode := L_MC4P_Orientation_Mode.ShortestSpacialWay;
	AEDIRECTION : ARRAY [4..6] OF MC_DIRECTION := [3(MC_DIRECTION.mcShortestWay)];
END_VAR
VAR_OUTPUT
	XDONE : BOOL;
	XBUSY : BOOL;
	XACTIVE : BOOL;
	XCOMMANDABORTED : BOOL;
	XERROR : BOOL;
	EERRORID : L_IE1P_Error;
END_VAR
VAR
	ECIRCMODE : L_MC4P_CircMode := L_MC4P_CircMode.CENTER;
	CLASSID : DINT;
END_VAR
END_FUNCTION_BLOCK

METHOD HOMINGREQUIRED : BOOL
END_METHOD

METHOD MAIN
VAR_IN_OUT
	AXESGROUP : AXES_GROUP_KIN;
	FBBASE : L_MC4P_Template_AG_KIN;
END_VAR
END_METHOD

METHOD PARAMETERFREEZE
VAR_IN_OUT
	AXESGROUP : AXES_GROUP_KIN;
	FBBASE : L_MC4P_Template_AG_KIN;
	COORDSYSTEM : L_MC4P_CoordSystem;
	BUFFERMODE : MC_BUFFER_MODE;
	TRANSITIONMODE : MC_TRANSITION_MODE;
	TRANSITIONPARAMETER : ARRAY [1..12] OF LREAL;
END_VAR
END_METHOD

METHOD SETERRORINPUTLIMITATIONVIOLATION
VAR_IN_OUT
	FBBASE : L_MC4P_Template_AG_KIN;
END_VAR
END_METHOD

METHOD SETPATHELEMENT
VAR_IN_OUT
	AXESGROUP : AXES_GROUP_KIN;
	FBBASE : L_MC4P_Template_AG_KIN;
	ALRSTARTPOS : ARRAY [1..12] OF LREAL;
	ALRSUPERPOSPOSATSTART : ARRAY [1..3] OF LREAL;
END_VAR
END_METHOD

METHOD FB_INIT : BOOL
VAR_INPUT
	BINITRETAINS : BOOL;
	BINCOPYCODE : BOOL;
END_VAR
END_METHOD

(* ---- L_MC4P_MOVEELLIPTICALABSOLUTEPNP.pou ---- *)
FUNCTION_BLOCK L_MC4P_MOVEELLIPTICALABSOLUTEPNP EXTENDS L_MC4P_Template_MoveLicence
VAR_INPUT
	XEXECUTE : BOOL;
	ALRENDPOINT : ARRAY [1..12] OF LREAL;
	ALRDIRECTION : ARRAY [1..3] OF LREAL;
	LRSEMIAXIS : LREAL;
	EELLIPTICALPNPMODE : L_MC4P_EllipticalPnPMode := L_MC4P_EllipticalPnPMode.Elliptical_180;
	LRVELOCITY : LREAL;
	LRACCELERATION : LREAL;
	LRDECELERATION : LREAL;
	LRJERK : LREAL;
	ECOORDSYSTEM : L_MC4P_CoordSystem;
	EBUFFERMODE : MC_BUFFER_MODE;
	ETRANSITIONMODE : MC_TRANSITION_MODE;
	ALRTRANSITIONPARAMETER : ARRAY [1..12] OF LREAL := [12(0)];
	AEAUXMODE : ARRAY [1..6] OF L_MC4P_AuxMode;
	EORIENTATIONMODE : L_MC4P_Orientation_Mode := L_MC4P_Orientation_Mode.ShortestSpacialWay;
	AEDIRECTION : ARRAY [4..6] OF MC_DIRECTION := [3(MC_DIRECTION.mcShortestWay)];
END_VAR
VAR_OUTPUT
	XDONE : BOOL;
	XBUSY : BOOL;
	XACTIVE : BOOL;
	XCOMMANDABORTED : BOOL;
	XERROR : BOOL;
	EERRORID : L_IE1P_Error;
END_VAR
VAR
	MOVEELLIPTICAL : L_MC4P_MoveEllipticalAbsolutePnP_Internal;
	PMOVE : POINTER TO L_MC4P_MoveContPath;
END_VAR
END_FUNCTION_BLOCK

(* ---- L_MC4P_MOVEELLIPTICALABSOLUTEPNP_INTERNAL.pou ---- *)
FUNCTION_BLOCK L_MC4P_MOVEELLIPTICALABSOLUTEPNP_INTERNAL EXTENDS L_MC4P_MoveContPath
VAR_INPUT
	XEXECUTE : BOOL;
	ALRENDPOINT : ARRAY [1..12] OF LREAL;
	ALRDIRECTION : ARRAY [1..3] OF LREAL;
	LRSEMIAXIS : LREAL;
	EELLIPTICALPNPMODE : L_MC4P_EllipticalPnPMode := L_MC4P_EllipticalPnPMode.Elliptical_180;
	LRVELOCITY : LREAL;
	LRACCELERATION : LREAL;
	LRDECELERATION : LREAL;
	LRJERK : LREAL;
	ECOORDSYSTEM : L_MC4P_CoordSystem;
	EBUFFERMODE : MC_BUFFER_MODE;
	ETRANSITIONMODE : MC_TRANSITION_MODE;
	ALRTRANSITIONPARAMETER : ARRAY [1..12] OF LREAL := [12(0)];
	AEAUXMODE : ARRAY [1..6] OF L_MC4P_AuxMode;
	EORIENTATIONMODE : L_MC4P_Orientation_Mode := L_MC4P_Orientation_Mode.ShortestSpacialWay;
	AEDIRECTION : ARRAY [4..6] OF MC_DIRECTION := [3(MC_DIRECTION.mcShortestWay)];
END_VAR
VAR_OUTPUT
	XDONE : BOOL;
	XBUSY : BOOL;
	XACTIVE : BOOL;
	XCOMMANDABORTED : BOOL;
	XERROR : BOOL;
	EERRORID : L_IE1P_Error;
END_VAR
VAR
	ECIRCMODE : L_MC4P_CircMode := L_MC4P_CircMode.CENTER;
	EPATHCHOICE : MC_CIRC_PATHCHOICE := MC_CIRC_PATHCHOICE.CLOCKWISE;
	CLASSID : DINT;
END_VAR
END_FUNCTION_BLOCK

METHOD HOMINGREQUIRED : BOOL
END_METHOD

METHOD MAIN
VAR_IN_OUT
	AXESGROUP : AXES_GROUP_KIN;
	FBBASE : L_MC4P_Template_AG_KIN;
END_VAR
END_METHOD

METHOD PARAMETERFREEZE
VAR_IN_OUT
	AXESGROUP : AXES_GROUP_KIN;
	FBBASE : L_MC4P_Template_AG_KIN;
	COORDSYSTEM : L_MC4P_CoordSystem;
	BUFFERMODE : MC_BUFFER_MODE;
	TRANSITIONMODE : MC_TRANSITION_MODE;
	TRANSITIONPARAMETER : ARRAY [1..12] OF LREAL;
END_VAR
END_METHOD

METHOD SETERRORINPUTLIMITATIONVIOLATION
VAR_IN_OUT
	FBBASE : L_MC4P_Template_AG_KIN;
END_VAR
END_METHOD

METHOD SETPATHELEMENT
VAR_IN_OUT
	AXESGROUP : AXES_GROUP_KIN;
	FBBASE : L_MC4P_Template_AG_KIN;
	ALRSTARTPOS : ARRAY [1..12] OF LREAL;
	ALRSUPERPOSPOSATSTART : ARRAY [1..3] OF LREAL;
END_VAR
END_METHOD

METHOD FB_INIT : BOOL
VAR_INPUT
	BINITRETAINS : BOOL;
	BINCOPYCODE : BOOL;
END_VAR
END_METHOD

(* ---- L_MC4P_MOVEELLIPTICALRELATIVE.pou ---- *)
FUNCTION_BLOCK L_MC4P_MOVEELLIPTICALRELATIVE EXTENDS L_MC4P_Template_MoveLicence
VAR_INPUT
	XEXECUTE : BOOL;
	ALRAUXPOINT : ARRAY [1..12] OF LREAL;
	ALRENDPOINT : ARRAY [1..12] OF LREAL;
	LRSEMIMAJORAXIS : LREAL;
	LRSEMIMINORAXIS : LREAL;
	EPATHCHOICE : MC_CIRC_PATHCHOICE;
	LRVELOCITY : LREAL;
	LRACCELERATION : LREAL;
	LRDECELERATION : LREAL;
	LRJERK : LREAL;
	ECOORDSYSTEM : L_MC4P_CoordSystem;
	EBUFFERMODE : MC_BUFFER_MODE;
	ETRANSITIONMODE : MC_TRANSITION_MODE;
	ALRTRANSITIONPARAMETER : ARRAY [1..12] OF LREAL := [12(0)];
	AEAUXMODE : ARRAY [1..6] OF L_MC4P_AuxMode;
	EORIENTATIONMODE : L_MC4P_Orientation_Mode := L_MC4P_Orientation_Mode.ShortestSpacialWay;
	AEDIRECTION : ARRAY [4..6] OF MC_DIRECTION := [3(MC_DIRECTION.mcShortestWay)];
END_VAR
VAR_OUTPUT
	XDONE : BOOL;
	XBUSY : BOOL;
	XACTIVE : BOOL;
	XCOMMANDABORTED : BOOL;
	XERROR : BOOL;
	EERRORID : L_IE1P_Error;
END_VAR
VAR
	MOVEELLIPTICAL : L_MC4P_MoveEllipticalRelative_Internal;
	PMOVE : POINTER TO L_MC4P_MoveContPath;
	SETELLIPTICALTARGETTOLERANCE : LREAL;
END_VAR
END_FUNCTION_BLOCK

(* ---- L_MC4P_MOVEELLIPTICALRELATIVE_INTERNAL.pou ---- *)
FUNCTION_BLOCK L_MC4P_MOVEELLIPTICALRELATIVE_INTERNAL EXTENDS L_MC4P_MoveContPath
VAR_INPUT
	XEXECUTE : BOOL;
	ALRAUXPOINT : ARRAY [1..12] OF LREAL;
	ALRENDPOINT : ARRAY [1..12] OF LREAL;
	LRSEMIMAJORAXIS : LREAL;
	LRSEMIMINORAXIS : LREAL;
	EPATHCHOICE : MC_CIRC_PATHCHOICE;
	LRVELOCITY : LREAL;
	LRACCELERATION : LREAL;
	LRDECELERATION : LREAL;
	LRJERK : LREAL;
	ECOORDSYSTEM : L_MC4P_CoordSystem;
	EBUFFERMODE : MC_BUFFER_MODE;
	ETRANSITIONMODE : MC_TRANSITION_MODE;
	ALRTRANSITIONPARAMETER : ARRAY [1..12] OF LREAL := [12(0)];
	AEAUXMODE : ARRAY [1..6] OF L_MC4P_AuxMode;
	EORIENTATIONMODE : L_MC4P_Orientation_Mode := L_MC4P_Orientation_Mode.ShortestSpacialWay;
	AEDIRECTION : ARRAY [4..6] OF MC_DIRECTION := [3(MC_DIRECTION.mcShortestWay)];
END_VAR
VAR_OUTPUT
	XDONE : BOOL;
	XBUSY : BOOL;
	XACTIVE : BOOL;
	XCOMMANDABORTED : BOOL;
	XERROR : BOOL;
	EERRORID : L_IE1P_Error;
END_VAR
VAR
	ECIRCMODE : L_MC4P_CircMode := L_MC4P_CircMode.CENTER;
	CLASSID : DINT;
END_VAR
END_FUNCTION_BLOCK

METHOD HOMINGREQUIRED : BOOL
END_METHOD

METHOD MAIN
VAR_IN_OUT
	AXESGROUP : AXES_GROUP_KIN;
	FBBASE : L_MC4P_Template_AG_KIN;
END_VAR
END_METHOD

METHOD PARAMETERFREEZE
VAR_IN_OUT
	AXESGROUP : AXES_GROUP_KIN;
	FBBASE : L_MC4P_Template_AG_KIN;
	COORDSYSTEM : L_MC4P_CoordSystem;
	BUFFERMODE : MC_BUFFER_MODE;
	TRANSITIONMODE : MC_TRANSITION_MODE;
	TRANSITIONPARAMETER : ARRAY [1..12] OF LREAL;
END_VAR
END_METHOD

METHOD SETERRORINPUTLIMITATIONVIOLATION
VAR_IN_OUT
	FBBASE : L_MC4P_Template_AG_KIN;
END_VAR
END_METHOD

METHOD SETPATHELEMENT
VAR_IN_OUT
	AXESGROUP : AXES_GROUP_KIN;
	FBBASE : L_MC4P_Template_AG_KIN;
	ALRSTARTPOS : ARRAY [1..12] OF LREAL;
	ALRSUPERPOSPOSATSTART : ARRAY [1..3] OF LREAL;
END_VAR
END_METHOD

METHOD FB_INIT : BOOL
VAR_INPUT
	BINITRETAINS : BOOL;
	BINCOPYCODE : BOOL;
END_VAR
END_METHOD

(* ---- L_MC4P_MOVEFBDIAGNOSTIC.pou ---- *)
FUNCTION_BLOCK L_MC4P_MOVEFBDIAGNOSTIC
VAR_INPUT
	XEXECUTEWRITETEXTFILE : BOOL;
	XENABLE : BOOL;
END_VAR
VAR_OUTPUT
	XWRITEFILEDONE : BOOL;
	XWRITEFILEBUSY : BOOL;
	XWRITEFILEERROR : BOOL;
	XBUSY : BOOL;
END_VAR
VAR
	ASCPARAMS : ARRAY [0..wDepth] OF L_MC4P_Parameter_MCMove;
	ADWTIMESTAMP : ARRAY [0..wDepth] OF DWORD;
	ASINSTANCESTR : ARRAY [0..wDepth] OF STRING;
	WCURRENTPOS : WORD := 0;
	SCPARAMDUMMY : L_MC4P_Parameter_MCMove;
	XTESTINMOTIONTASK : BOOL := FALSE;
	XFREETASKBUSY_INT : BOOL;
	XFREETASKDONE_INT : BOOL;
	XFREETASKERROR_INT : BOOL;
	EFREETASKEERRORID_INT : L_IE1P_Error;
	XEXECUTEWRITETEXTFILE_OLD : BOOL;
	SEXCELFILENAME : STRING(255);
	RES : SYSFILE.RTS_IEC_ResULT;
	HFILE : SYSFILE.RTS_IEC_HANDLE;
	XWFSIZE : __XWORD;
	XWRESULTWRITESTRING : __XWORD;
	ASHEADLINEPARAMS : ARRAY [1..iMaxHeadLine] OF STRING := ['TimeStamp', 'sInstanceStr', 'SegmentType', 'xMoveRel', 'Position', 'Distance', 'CircMode', 'AuxPoint', 'PathChoice', 'lrSemiMajorAxis', 'lrSemiMinorAxis', 'ascIntermediatePointSpline', 'Velocity', 'Acceleration', 'Deceleration', 'Jerk', 'alrVelocityPTP', 'alrAccelerationPTP', 'alrDecelerationPTP', 'alrJerkPTP', 'alrVelocityAux', 'alrAccelerationAux', 'alrDecelerationAux', 'alrJerkAux', 'CoordSystem', 'CoordRef', 'BufferMode', 'TransitionMode', 'TransitionParameter', 'aeAuxMode', 'alrAxisLimitVel', 'alrAxisLimitAcc', 'alrAxisLimitJerk', 'aiTargetConfiguration', 'eOrientationMode', 'aeDirection'];
	STABULATOR : STRING(2) := '$T';
	SLINEFEED : STRING(2) := '$N';
	SZEILE : STRING(255);
	WSTEPWF : WORD := 0;
	XAGERROR : BOOL;
	WLOOKAHEADHORIZON : WORD;
	DWTASKCYCLE_US : DWORD;
	EACTIVEERRORID : L_IE1P_Error;
	SAXESGROUPNAME : STRING;
	VERSION : VERSION;
	WDEPTH : WORD := 50;
	IMAXHEADLINE : INT := 40;
	ACTIVEERRORID : WORD;
	AGERROR : BOOL;
	AXESGROUPNAME : STRING;
	LOOKAHEADHORIZON : WORD;
	TASKCYCLE_US : DWORD;
	VERSIONMC4P : VERSION;
	XWRITEINMOTIONTASK : BOOL;
END_VAR
END_FUNCTION_BLOCK

METHOD FREEZEMOVEFBPARAM
VAR_INPUT
	SINSTANCESTR : STRING;
	DWTIMESTAMP : DWORD;
END_VAR
VAR_IN_OUT
	INPUT_PARAMETER : L_MC4P_Parameter_MCMove;
END_VAR
END_METHOD

METHOD FREEZESTOPALLPARAM
VAR_INPUT
	SINSTANCESTR : STRING;
	DWTIMESTAMP : DWORD;
END_VAR
VAR_IN_OUT
	ASCCTRLABC : ARRAY [1..18] OF L_MC1P_CtrlABC;
END_VAR
END_METHOD

METHOD FREEZESTOPPARAM
VAR_INPUT
	SINSTANCESTR : STRING;
	DWTIMESTAMP : DWORD;
	LRINPUTDECELERATION : LREAL;
	LRINPUTJERK : LREAL;
END_VAR
END_METHOD

METHOD CALL_WRITEEXCELFILE
END_METHOD

METHOD EXECUTEFREERUNTASK
VAR_INPUT
	SDIR : STRING;
END_VAR
END_METHOD

METHOD MAIN
END_METHOD

METHOD ABORT : UDINT
END_METHOD

METHOD EXECUTE : UDINT
END_METHOD

(* ---- L_MC4P_MOVEFBPOOL.pou ---- *)
FUNCTION_BLOCK L_MC4P_MOVEFBPOOL EXTENDS L_UBUP_FBPool
VAR
	_PICKANDPLACEMEMORY : REFERENCE TO L_MC4P_PickAndPlaceMemory;
	_XMEMOWNER1 : BOOL;
	_SCFBSTORE : REFERENCE TO L_MC4P_MovePathStore;
	_XMEMOWNER2 : BOOL;
	_AFB_MOVEELLIPTICALABS : ARRAY [1..3] OF L_MC4P_MoveEllipticalAbsolute_Internal;
	_MOVELINABSCONTROLNODES : L_UBUP_DoubleLinkedListNodes;
	_MOVELINABSCONTROL : L_UBUP_DoubleLinkedListControl;
	_MOVELINRELCONTROLNODES : L_UBUP_DoubleLinkedListNodes;
	_MOVELINRELCONTROL : L_UBUP_DoubleLinkedListControl;
	_MOVEDIRABSCONTROLNODES : L_UBUP_DoubleLinkedListNodes;
	_MOVEDIRABSCONTROL : L_UBUP_DoubleLinkedListControl;
	_MOVEDIRRELCONTROLNODES : L_UBUP_DoubleLinkedListNodes;
	_MOVEDIRRELCONTROL : L_UBUP_DoubleLinkedListControl;
	_MOVEELLIPTPNPCONTROLNODES : L_UBUP_DoubleLinkedListNodes;
	_MOVEELLIPTPNPCONTROL : L_UBUP_DoubleLinkedListControl;
	_MOVEELLIPTABSCONTROLNODES : L_UBUP_DoubleLinkedListNodes;
	_MOVEELLIPTABSCONTROL : L_UBUP_DoubleLinkedListControl;
	_MOVESPLINEPNPCONTROLNODES : L_UBUP_DoubleLinkedListNodes;
	_MOVESPLINEPNPCONTROL : L_UBUP_DoubleLinkedListControl;
	_MOVECONTPATHCONTROLNODES : L_UBUP_DoubleLinkedListNodes;
	_MOVECONTPATHCONTROL : L_UBUP_DoubleLinkedListControl;
	USEGLOBAL : BOOL;
END_VAR
END_FUNCTION_BLOCK

METHOD FREEINSTANCE : BOOL
VAR_INPUT
	ITFINSTANCE : L_UBUP_IPoolInstance;
	XWHANDLE : __XWORD;
END_VAR
END_METHOD

METHOD GETCAPACITY : BOOL
VAR_INPUT
	ECLASSID : DINT;
END_VAR
VAR_OUTPUT
	DWCAPACITY : DWORD;
END_VAR
END_METHOD

METHOD QUERYINSTANCE : BOOL
VAR_INPUT
	ECLASSID : DINT;
END_VAR
VAR_IN_OUT
	ITFINSTANCE : L_UBUP_IPoolInstance;
END_VAR
END_METHOD

METHOD FB_INIT : BOOL
VAR_INPUT
	BINITRETAINS : BOOL;
	BINCOPYCODE : BOOL;
END_VAR
END_METHOD

METHOD FB_AFTERGLOBALINIT : BOOL
END_METHOD

METHOD FREERESOURCE
END_METHOD

METHOD GETFB : L_UBUP_IPoolInstance
VAR_INPUT
	ECLASSID : DINT;
	DWARRIDX : DWORD;
END_VAR
END_METHOD

METHOD GETFBCONTROL : L_UBUP_IListControl
VAR_INPUT
	ECLASSID : DINT;
END_VAR
END_METHOD

METHOD OCCUPYRESOURCE : BOOL
VAR_INPUT
	ECLASSID : DINT;
END_VAR
END_METHOD

METHOD SETCAPACITY
VAR_INPUT
	ITFLISTCONTROL : L_UBUP_IListControl;
	DWCAPACITY : DWORD;
END_VAR
END_METHOD

METHOD SETCAPACITYALL
END_METHOD

METHOD FB_INIT : BOOL
VAR_INPUT
	BINITRETAINS : BOOL;
	BINCOPYCODE : BOOL;
	PICKANDPLACEMEMORY : REFERENCE TO L_MC4P_PickAndPlaceMemory;
	SCFBSTORE : REFERENCE TO L_MC4P_MovePathStore;
END_VAR
END_METHOD

METHOD FREERESOURCE
END_METHOD

METHOD GETFB : L_UBUP_IPoolInstance
VAR_INPUT
	ECLASSID : DINT;
	DWARRIDX : DWORD;
END_VAR
END_METHOD

METHOD GETFBCONTROL : L_UBUP_IListControl
VAR_INPUT
	ECLASSID : DINT;
END_VAR
END_METHOD

METHOD OCCUPYRESOURCE : BOOL
VAR_INPUT
	ECLASSID : DINT;
END_VAR
END_METHOD

METHOD SETCAPACITYALL
END_METHOD

(* ---- L_MC4P_MOVELINEARABSOLUTE_INTERNAL.pou ---- *)
FUNCTION_BLOCK L_MC4P_MOVELINEARABSOLUTE_INTERNAL EXTENDS L_MC4P_MoveContPath
VAR_INPUT
	EXECUTE : BOOL;
	POSITION : ARRAY [1..12] OF LREAL;
	VELOCITY : LREAL;
	ACCELERATION : LREAL;
	DECELERATION : LREAL;
	JERK : LREAL;
	COORDSYSTEM : L_MC4P_CoordSystem;
	BUFFERMODE : MC_BUFFER_MODE;
	TRANSITIONMODE : MC_TRANSITION_MODE;
	TRANSITIONPARAMETER : ARRAY [1..12] OF LREAL := [12(0)];
	AEAUXMODE : ARRAY [1..6] OF L_MC4P_AuxMode;
	ORIENTATIONMODE : L_MC4P_Orientation_Mode := L_MC4P_Orientation_Mode.ShortestSpacialWay;
	DIRECTION : ARRAY [4..6] OF MC_DIRECTION := [3(MC_DIRECTION.mcShortestWay)];
END_VAR
VAR_OUTPUT
	DONE : BOOL;
	BUSY : BOOL;
	ACTIVE : BOOL;
	COMMANDABORTED : BOOL;
	ERROR : BOOL;
	ERRORID : L_IE1P_Error;
END_VAR
VAR
	CLASSID : DINT;
END_VAR
END_FUNCTION_BLOCK

METHOD HOMINGREQUIRED : BOOL
END_METHOD

METHOD MAIN
VAR_IN_OUT
	AXESGROUP : AXES_GROUP_KIN;
	FBBASE : L_MC4P_Template_AG_KIN;
END_VAR
END_METHOD

METHOD PARAMETERFREEZE
VAR_IN_OUT
	AXESGROUP : AXES_GROUP_KIN;
	FBBASE : L_MC4P_Template_AG_KIN;
	COORDSYSTEM : L_MC4P_CoordSystem;
	BUFFERMODE : MC_BUFFER_MODE;
	TRANSITIONMODE : MC_TRANSITION_MODE;
	TRANSITIONPARAMETER : ARRAY [1..12] OF LREAL;
END_VAR
END_METHOD

METHOD SETERRORINPUTLIMITATIONVIOLATION
VAR_IN_OUT
	FBBASE : L_MC4P_Template_AG_KIN;
END_VAR
END_METHOD

METHOD SETPATHELEMENT
VAR_IN_OUT
	AXESGROUP : AXES_GROUP_KIN;
	FBBASE : L_MC4P_Template_AG_KIN;
	ALRSTARTPOS : ARRAY [1..12] OF LREAL;
	ALRSUPERPOSPOSATSTART : ARRAY [1..3] OF LREAL;
END_VAR
END_METHOD

(* ---- L_MC4P_MOVELINEARRELATIVE_INTERNAL.pou ---- *)
FUNCTION_BLOCK L_MC4P_MOVELINEARRELATIVE_INTERNAL EXTENDS L_MC4P_MoveContPath
VAR_INPUT
	EXECUTE : BOOL;
	DISTANCE : ARRAY [1..12] OF LREAL;
	VELOCITY : LREAL;
	ACCELERATION : LREAL;
	DECELERATION : LREAL;
	JERK : LREAL;
	COORDSYSTEM : L_MC4P_CoordSystem;
	BUFFERMODE : MC_BUFFER_MODE;
	TRANSITIONMODE : MC_TRANSITION_MODE;
	TRANSITIONPARAMETER : ARRAY [1..12] OF LREAL := [12(0)];
	AEAUXMODE : ARRAY [1..6] OF L_MC4P_AuxMode;
	ORIENTATIONMODE : L_MC4P_Orientation_Mode := L_MC4P_Orientation_Mode.ShortestSpacialWay;
	DIRECTION : ARRAY [4..6] OF MC_DIRECTION := [3(MC_DIRECTION.mcShortestWay)];
END_VAR
VAR_OUTPUT
	DONE : BOOL;
	BUSY : BOOL;
	ACTIVE : BOOL;
	COMMANDABORTED : BOOL;
	ERROR : BOOL;
	ERRORID : L_IE1P_Error;
END_VAR
VAR
	CLASSID : DINT;
END_VAR
END_FUNCTION_BLOCK

METHOD HOMINGREQUIRED : BOOL
END_METHOD

METHOD MAIN
VAR_IN_OUT
	AXESGROUP : AXES_GROUP_KIN;
	FBBASE : L_MC4P_Template_AG_KIN;
END_VAR
END_METHOD

METHOD PARAMETERFREEZE
VAR_IN_OUT
	AXESGROUP : AXES_GROUP_KIN;
	FBBASE : L_MC4P_Template_AG_KIN;
	COORDSYSTEM : L_MC4P_CoordSystem;
	BUFFERMODE : MC_BUFFER_MODE;
	TRANSITIONMODE : MC_TRANSITION_MODE;
	TRANSITIONPARAMETER : ARRAY [1..12] OF LREAL;
END_VAR
END_METHOD

METHOD SETERRORINPUTLIMITATIONVIOLATION
VAR_IN_OUT
	FBBASE : L_MC4P_Template_AG_KIN;
END_VAR
END_METHOD

METHOD SETPATHELEMENT
VAR_IN_OUT
	AXESGROUP : AXES_GROUP_KIN;
	FBBASE : L_MC4P_Template_AG_KIN;
	ALRSTARTPOS : ARRAY [1..12] OF LREAL;
	ALRSUPERPOSPOSATSTART : ARRAY [1..3] OF LREAL;
END_VAR
END_METHOD

(* ---- L_MC4P_MOVESPLINEABSOLUTE.pou ---- *)
FUNCTION_BLOCK L_MC4P_MOVESPLINEABSOLUTE EXTENDS L_MC4P_Template_MoveLicence
VAR_INPUT
	XEXECUTE : BOOL;
	ASCINTERMEDIATEPOINT : ARRAY [1..9] OF L_MC4P_IntermediatePointSpline;
	ALRENDPOINT : ARRAY [1..12] OF LREAL;
	LRVELOCITY : LREAL;
	LRACCELERATION : LREAL;
	LRDECELERATION : LREAL;
	LRJERK : LREAL;
	ECOORDSYSTEM : L_MC4P_CoordSystem;
	EBUFFERMODE : MC_BUFFER_MODE;
	ETRANSITIONMODE : MC_TRANSITION_MODE;
	ALRTRANSITIONPARAMETER : ARRAY [1..12] OF LREAL := [12(0)];
	AEAUXMODE : ARRAY [1..6] OF L_MC4P_AuxMode;
	EORIENTATIONMODE : L_MC4P_Orientation_Mode := L_MC4P_Orientation_Mode.ShortestSpacialWay;
	AEDIRECTION : ARRAY [4..6] OF MC_DIRECTION := [3(MC_DIRECTION.mcShortestWay)];
END_VAR
VAR_OUTPUT
	XDONE : BOOL;
	XBUSY : BOOL;
	XACTIVE : BOOL;
	XCOMMANDABORTED : BOOL;
	XERROR : BOOL;
	EERRORID : L_IE1P_Error;
	IPOINTPASSED : INT;
END_VAR
VAR
	MOVESPLINE : L_MC4P_MoveSplineAbsolute_Internal;
	XDIALOGINTERMEDIATEPOINT : BOOL := FALSE;
	IVISUTABLESETPOS : INT := 1;
	PASSEDINTERMEDIATEPOINT : INT;
	PMOVE : POINTER TO L_MC4P_MoveContPath;
END_VAR
END_FUNCTION_BLOCK

(* ---- L_MC4P_MOVESPLINEABSOLUTE_INTERNAL.pou ---- *)
FUNCTION_BLOCK L_MC4P_MOVESPLINEABSOLUTE_INTERNAL EXTENDS L_MC4P_MoveContPath
VAR_INPUT
	XEXECUTE : BOOL;
	ASCINTERMEDIATEPOINT : ARRAY [1..9] OF L_MC4P_IntermediatePointSpline;
	ALRENDPOINT : ARRAY [1..12] OF LREAL;
	LRVELOCITY : LREAL;
	LRACCELERATION : LREAL;
	LRDECELERATION : LREAL;
	LRJERK : LREAL;
	ECOORDSYSTEM : L_MC4P_CoordSystem;
	EBUFFERMODE : MC_BUFFER_MODE;
	ETRANSITIONMODE : MC_TRANSITION_MODE;
	ALRTRANSITIONPARAMETER : ARRAY [1..12] OF LREAL := [12(0)];
	AEAUXMODE : ARRAY [1..6] OF L_MC4P_AuxMode;
	EORIENTATIONMODE : L_MC4P_Orientation_Mode := L_MC4P_Orientation_Mode.ShortestSpacialWay;
	AEDIRECTION : ARRAY [4..6] OF MC_DIRECTION := [3(MC_DIRECTION.mcShortestWay)];
END_VAR
VAR_OUTPUT
	XDONE : BOOL;
	XBUSY : BOOL;
	XACTIVE : BOOL;
	XCOMMANDABORTED : BOOL;
	XERROR : BOOL;
	EERRORID : L_IE1P_Error;
	IPOINTPASSED : INT;
END_VAR
VAR
	CLASSID : DINT;
	PASSEDINTERMEDIATEPOINT : INT;
END_VAR
END_FUNCTION_BLOCK

METHOD HOMINGREQUIRED : BOOL
END_METHOD

METHOD MAIN
VAR_IN_OUT
	AXESGROUP : AXES_GROUP_KIN;
	FBBASE : L_MC4P_Template_AG_KIN;
END_VAR
END_METHOD

METHOD PARAMETERFREEZE
VAR_IN_OUT
	AXESGROUP : AXES_GROUP_KIN;
	FBBASE : L_MC4P_Template_AG_KIN;
	COORDSYSTEM : L_MC4P_CoordSystem;
	BUFFERMODE : MC_BUFFER_MODE;
	TRANSITIONMODE : MC_TRANSITION_MODE;
	TRANSITIONPARAMETER : ARRAY [1..12] OF LREAL;
END_VAR
END_METHOD

METHOD SETERRORINPUTLIMITATIONVIOLATION
VAR_IN_OUT
	FBBASE : L_MC4P_Template_AG_KIN;
END_VAR
END_METHOD

METHOD SETPATHELEMENT
VAR_IN_OUT
	AXESGROUP : AXES_GROUP_KIN;
	FBBASE : L_MC4P_Template_AG_KIN;
	ALRSTARTPOS : ARRAY [1..12] OF LREAL;
	ALRSUPERPOSPOSATSTART : ARRAY [1..3] OF LREAL;
END_VAR
END_METHOD

(* ---- L_MC4P_MOVESPLINEPNP.pou ---- *)
FUNCTION_BLOCK L_MC4P_MOVESPLINEPNP EXTENDS L_MC4P_Template_MoveLicence
VAR_INPUT
	XEXECUTE : BOOL;
	LRZSTARTDIST : LREAL;
	LRZTARGETDIST : LREAL;
	ALRENDPOINT : ARRAY [1..12] OF LREAL;
	LRZMAXHEIGHT : LREAL;
	LRVELOCITY : LREAL;
	LRACCELERATION : LREAL;
	LRDECELERATION : LREAL;
	LRJERK : LREAL;
	ECOORDSYSTEM : L_MC4P_CoordSystem;
	EBUFFERMODE : MC_BUFFER_MODE;
	ETRANSITIONMODE : MC_TRANSITION_MODE;
	ALRTRANSITIONPARAMETER : ARRAY [1..12] OF LREAL := [12(0)];
	AEAUXMODE : ARRAY [1..6] OF L_MC4P_AuxMode;
	EORIENTATIONMODE : L_MC4P_Orientation_Mode := L_MC4P_Orientation_Mode.ShortestSpacialWay;
	AEDIRECTION : ARRAY [4..6] OF MC_DIRECTION := [3(MC_DIRECTION.mcShortestWay)];
END_VAR
VAR_OUTPUT
	XDONE : BOOL;
	XBUSY : BOOL;
	XACTIVE : BOOL;
	XCOMMANDABORTED : BOOL;
	XERROR : BOOL;
	EERRORID : L_IE1P_Error;
	IPOINTPASSED : INT;
END_VAR
VAR
	MOVESPLINE : L_MC4P_MoveSplinePnP_Internal;
	PASSEDINTERMEDIATEPOINT : INT;
	PMOVE : POINTER TO L_MC4P_MoveContPath;
END_VAR
END_FUNCTION_BLOCK

(* ---- L_MC4P_MOVESPLINEPNP_INTERNAL.pou ---- *)
FUNCTION_BLOCK L_MC4P_MOVESPLINEPNP_INTERNAL EXTENDS L_MC4P_MoveContPath
VAR_INPUT
	XEXECUTE : BOOL;
	LRZSTARTDIST : LREAL;
	LRZTARGETDIST : LREAL;
	ALRENDPOINT : ARRAY [1..12] OF LREAL;
	LRZMAXHEIGHT : LREAL;
	LRVELOCITY : LREAL;
	LRACCELERATION : LREAL;
	LRDECELERATION : LREAL;
	LRJERK : LREAL;
	ECOORDSYSTEM : L_MC4P_CoordSystem;
	EBUFFERMODE : MC_BUFFER_MODE;
	ETRANSITIONMODE : MC_TRANSITION_MODE;
	ALRTRANSITIONPARAMETER : ARRAY [1..12] OF LREAL := [12(0)];
	AEAUXMODE : ARRAY [1..6] OF L_MC4P_AuxMode;
	EORIENTATIONMODE : L_MC4P_Orientation_Mode := L_MC4P_Orientation_Mode.ShortestSpacialWay;
	AEDIRECTION : ARRAY [4..6] OF MC_DIRECTION := [3(MC_DIRECTION.mcShortestWay)];
END_VAR
VAR_OUTPUT
	XDONE : BOOL;
	XBUSY : BOOL;
	XACTIVE : BOOL;
	XCOMMANDABORTED : BOOL;
	XERROR : BOOL;
	EERRORID : L_IE1P_Error;
	IPOINTPASSED : INT;
END_VAR
VAR
	CLASSID : DINT;
	PASSEDINTERMEDIATEPOINT : INT;
END_VAR
END_FUNCTION_BLOCK

METHOD HOMINGREQUIRED : BOOL
END_METHOD

METHOD MAIN
VAR_IN_OUT
	AXESGROUP : AXES_GROUP_KIN;
	FBBASE : L_MC4P_Template_AG_KIN;
END_VAR
END_METHOD

METHOD PARAMETERFREEZE
VAR_IN_OUT
	AXESGROUP : AXES_GROUP_KIN;
	FBBASE : L_MC4P_Template_AG_KIN;
	COORDSYSTEM : L_MC4P_CoordSystem;
	BUFFERMODE : MC_BUFFER_MODE;
	TRANSITIONMODE : MC_TRANSITION_MODE;
	TRANSITIONPARAMETER : ARRAY [1..12] OF LREAL;
END_VAR
END_METHOD

METHOD SETERRORINPUTLIMITATIONVIOLATION
VAR_IN_OUT
	FBBASE : L_MC4P_Template_AG_KIN;
END_VAR
END_METHOD

METHOD SETPATHELEMENT
VAR_IN_OUT
	AXESGROUP : AXES_GROUP_KIN;
	FBBASE : L_MC4P_Template_AG_KIN;
	ALRSTARTPOS : ARRAY [1..12] OF LREAL;
	ALRSUPERPOSPOSATSTART : ARRAY [1..3] OF LREAL;
END_VAR
END_METHOD

(* ---- L_MC4P_MOVESPLINERELATIVE.pou ---- *)
FUNCTION_BLOCK L_MC4P_MOVESPLINERELATIVE EXTENDS L_MC4P_Template_MoveLicence
VAR_INPUT
	XEXECUTE : BOOL;
	ASCINTERMEDIATEPOINT : ARRAY [1..9] OF L_MC4P_IntermediatePointSpline;
	ALRENDPOINT : ARRAY [1..12] OF LREAL;
	LRVELOCITY : LREAL;
	LRACCELERATION : LREAL;
	LRDECELERATION : LREAL;
	LRJERK : LREAL;
	ECOORDSYSTEM : L_MC4P_CoordSystem;
	EBUFFERMODE : MC_BUFFER_MODE;
	ETRANSITIONMODE : MC_TRANSITION_MODE;
	ALRTRANSITIONPARAMETER : ARRAY [1..12] OF LREAL := [12(0)];
	AEAUXMODE : ARRAY [1..6] OF L_MC4P_AuxMode;
	EORIENTATIONMODE : L_MC4P_Orientation_Mode := L_MC4P_Orientation_Mode.ShortestSpacialWay;
	AEDIRECTION : ARRAY [4..6] OF MC_DIRECTION := [3(MC_DIRECTION.mcShortestWay)];
END_VAR
VAR_OUTPUT
	XDONE : BOOL;
	XBUSY : BOOL;
	XACTIVE : BOOL;
	XCOMMANDABORTED : BOOL;
	XERROR : BOOL;
	EERRORID : L_IE1P_Error;
	IPOINTPASSED : INT;
END_VAR
VAR
	MOVESPLINE : L_MC4P_MoveSplineRelative_Internal;
	XDIALOGINTERMEDIATEPOINT : BOOL := FALSE;
	IVISUTABLESETPOS : INT := 1;
	PASSEDINTERMEDIATEPOINT : INT;
	PMOVE : POINTER TO L_MC4P_MoveContPath;
END_VAR
END_FUNCTION_BLOCK

(* ---- L_MC4P_MOVESPLINERELATIVE_INTERNAL.pou ---- *)
FUNCTION_BLOCK L_MC4P_MOVESPLINERELATIVE_INTERNAL EXTENDS L_MC4P_MoveContPath
VAR_INPUT
	XEXECUTE : BOOL;
	ASCINTERMEDIATEPOINT : ARRAY [1..9] OF L_MC4P_IntermediatePointSpline;
	ALRENDPOINT : ARRAY [1..12] OF LREAL;
	LRVELOCITY : LREAL;
	LRACCELERATION : LREAL;
	LRDECELERATION : LREAL;
	LRJERK : LREAL;
	ECOORDSYSTEM : L_MC4P_CoordSystem;
	EBUFFERMODE : MC_BUFFER_MODE;
	ETRANSITIONMODE : MC_TRANSITION_MODE;
	ALRTRANSITIONPARAMETER : ARRAY [1..12] OF LREAL := [12(0)];
	AEAUXMODE : ARRAY [1..6] OF L_MC4P_AuxMode;
	EORIENTATIONMODE : L_MC4P_Orientation_Mode := L_MC4P_Orientation_Mode.ShortestSpacialWay;
	AEDIRECTION : ARRAY [4..6] OF MC_DIRECTION := [3(MC_DIRECTION.mcShortestWay)];
END_VAR
VAR_OUTPUT
	XDONE : BOOL;
	XBUSY : BOOL;
	XACTIVE : BOOL;
	XCOMMANDABORTED : BOOL;
	XERROR : BOOL;
	EERRORID : L_IE1P_Error;
	IPOINTPASSED : INT;
END_VAR
VAR
	CLASSID : DINT;
	PASSEDINTERMEDIATEPOINT : INT;
END_VAR
END_FUNCTION_BLOCK

METHOD HOMINGREQUIRED : BOOL
END_METHOD

METHOD MAIN
VAR_IN_OUT
	AXESGROUP : AXES_GROUP_KIN;
	FBBASE : L_MC4P_Template_AG_KIN;
END_VAR
END_METHOD

METHOD PARAMETERFREEZE
VAR_IN_OUT
	AXESGROUP : AXES_GROUP_KIN;
	FBBASE : L_MC4P_Template_AG_KIN;
	COORDSYSTEM : L_MC4P_CoordSystem;
	BUFFERMODE : MC_BUFFER_MODE;
	TRANSITIONMODE : MC_TRANSITION_MODE;
	TRANSITIONPARAMETER : ARRAY [1..12] OF LREAL;
END_VAR
END_METHOD

METHOD SETERRORINPUTLIMITATIONVIOLATION
VAR_IN_OUT
	FBBASE : L_MC4P_Template_AG_KIN;
END_VAR
END_METHOD

METHOD SETPATHELEMENT
VAR_IN_OUT
	AXESGROUP : AXES_GROUP_KIN;
	FBBASE : L_MC4P_Template_AG_KIN;
	ALRSTARTPOS : ARRAY [1..12] OF LREAL;
	ALRSUPERPOSPOSATSTART : ARRAY [1..3] OF LREAL;
END_VAR
END_METHOD

(* ---- L_MC4P_OBSERVELIMITS.pou ---- *)
FUNCTION_BLOCK L_MC4P_OBSERVELIMITS
VAR_INPUT
	XENABLE : BOOL;
	XRESETOBSERVEDLIMITS : BOOL;
	XHOLDOBSERVEDLIMITS : BOOL;
	PAXESGROUP : POINTER TO AXES_GROUP_KIN;
	UACTIVELIMITSMAN : L_MC1P.L_MC1P_uULINT;
END_VAR
VAR_OUTPUT
	UACTIVELIMITS : L_MC1P.L_MC1P_uULINT;
END_VAR
VAR
	XENABLEOLD : BOOL;
	IDX : INT;
	PAXIS : POINTER TO AXIS_REF;
	ALRSETACCOLD : ARRAY [1..6] OF LREAL;
	ALRSETJERK : ARRAY [1..6] OF LREAL;
	LRMAXVELFB : LREAL;
	LRMAXACCFB : LREAL;
	LRMAXJERKFB : LREAL;
	SCLAMPACTIVAX : ARRAY [1..12, 1..10, 0..1] OF BOOL;
	SCLAMPACTIVAG : ARRAY [1..3, 1..3, 0..1] OF BOOL;
	WVISUAXESFRAME : WORD;
	HEVENTCOMMCYCLE : Systypes.RTS_IEC_HANDLE := SysTypes.RTS_INVALID_HANDLE;
	HINTERFACECOMMCYCLE : Systypes.RTS_IEC_HANDLE := SysTypes.RTS_INVALID_HANDLE;
	ITFCALLBACK : CmpEventMgr.ICmpEventCallback;
	DWEVENTCOUNTER : DWORD;
END_VAR
END_FUNCTION_BLOCK

METHOD LIMITUSED : BOOL
VAR_INPUT
	LRCMPVAL : LREAL;
	LRACTVAL : LREAL;
END_VAR
END_METHOD

METHOD MAIN
END_METHOD

METHOD SETLAMPACTIV
END_METHOD

METHOD EVENTCALLBACK : UDINT
VAR_INPUT
	PEVENTPARAM : POINTER TO EventParam;
END_VAR
END_METHOD

METHOD REGISTEREVENT
END_METHOD

METHOD UNREGISTEREVENT
END_METHOD

(* ---- L_MC4P_PATHDATALIST.pou ---- *)
FUNCTION_BLOCK L_MC4P_PATHDATALIST
VAR_INPUT
	PAXESGROUP : POINTER TO AXES_GROUP_KIN;
END_VAR
VAR
	PLISTELEMENTFIRST : POINTER TO L_MC4P_ListElement;
	PLISTELEMENTLAST : POINTER TO L_MC4P_ListElement;
	XINITDONE : BOOL := FALSE;
	ARRLISTELEMENTS : ARRAY [0..L_MC4P_Constants.MaxCountListElements] OF L_MC4P_ListElement;
	SCINITIALLISTELEMENT : L_MC4P_ListElement;
END_VAR
END_FUNCTION_BLOCK

METHOD CALCPATHLENGTHLISTELEMENTS : LREAL
VAR_INPUT
	DWMASK : DWORD;
END_VAR
END_METHOD

METHOD CALCPATHLENGTHLISTELEMENTSOFFUNID : LREAL
VAR_INPUT
	DIFUNID : DINT;
END_VAR
END_METHOD

METHOD CALCTIMELISTELEMENTS : LREAL
VAR_INPUT
	DWMASK : DWORD;
END_VAR
END_METHOD

METHOD CALCTIMELISTELEMENTSOFFUNID : LREAL
VAR_INPUT
	DIFUNID : DINT;
END_VAR
END_METHOD

METHOD CHECKLIST : BOOL
END_METHOD

METHOD CHECKLISTANDPROFILES : BOOL
END_METHOD

METHOD CLEARFBPOINTER
VAR_INPUT
	PMOVECONTFB : POINTER TO L_MC4P_MoveContPath;
END_VAR
END_METHOD

METHOD COUNTLISTELEMENTS : INT
VAR_INPUT
	DWMASK : DWORD;
END_VAR
END_METHOD

METHOD DELETELISTELEMENT : BOOL
VAR_INPUT
	PLISTELEMENT : POINTER TO L_MC4P_ListElement;
END_VAR
END_METHOD

METHOD GETLISTELEMENTBYTIME : POINTER TO L_MC4P_ListElement
VAR_INPUT
	DWMASK : DWORD;
	LRTIMELISTIN : LREAL;
END_VAR
VAR_OUTPUT
	LRTIMEELEMENT : LREAL;
END_VAR
END_METHOD

METHOD GETLISTELEMENTOFFUNID : POINTER TO L_MC4P_ListElement
VAR_INPUT
	DIFUNID : DINT;
END_VAR
END_METHOD

METHOD GETNEWESTLISTELEMENT : POINTER TO L_MC4P_ListElement
VAR_INPUT
	DWMASK : DWORD;
END_VAR
END_METHOD

METHOD GETOLDESTLISTELEMENT : POINTER TO L_MC4P_ListElement
VAR_INPUT
	DWMASK : DWORD;
END_VAR
END_METHOD

METHOD GETOLDESTLISTELEMENTADVANCED : POINTER TO L_MC4P_ListElement
VAR_INPUT
	DWMASK : DWORD;
	DWPREVMASK : DWORD;
END_VAR
END_METHOD

METHOD INITLIST : BOOL
END_METHOD

METHOD INITLISTELEMENT : BOOL
VAR_INPUT
	PLISTELEMENT : POINTER TO L_MC4P_ListElement;
END_VAR
END_METHOD

METHOD INSERTLISTELEMENTBETWEEN : POINTER TO L_MC4P_ListElement
VAR_INPUT
	PPREVIOUS : POINTER TO L_MC4P_ListElement;
END_VAR
END_METHOD

METHOD INSERTNEWLISTELEMENT : POINTER TO L_MC4P_ListElement
END_METHOD

METHOD NUMLISTELEMENTSISLESSTHAN : BOOL
VAR_INPUT
	DWMASK : DWORD;
	IUPPER : INT;
END_VAR
END_METHOD

METHOD RESETLIST
END_METHOD

METHOD RESETMASKSINLIST
VAR_INPUT
	FIPOSECTIME : LREAL;
END_VAR
END_METHOD

METHOD STARTVELOFLISTELEMENTEQ0 : BOOL
VAR_INPUT
	PLISTELEMENT : POINTER TO L_MC4P_ListElement;
END_VAR
END_METHOD

METHOD TARGETVELOFLISTELEMENTEQ0 : BOOL
VAR_INPUT
	PLISTELEMENT : POINTER TO L_MC4P_ListElement;
END_VAR
END_METHOD

METHOD TIMELISTELEMENTSISLESSTHAN : BOOL
VAR_INPUT
	DWMASK : DWORD;
	LRUPPER : LREAL;
END_VAR
END_METHOD

METHOD _CREATELISTELEMENT : POINTER TO L_MC4P_ListElement
END_METHOD

METHOD _DESTROYLISTELEMENT
VAR_INPUT
	PLISTELEMENT : POINTER TO L_MC4P_ListElement;
END_VAR
END_METHOD

(* ---- L_MC4P_PATHLISTDIAGNOSTIC.pou ---- *)
FUNCTION_BLOCK L_MC4P_PATHLISTDIAGNOSTIC
VAR_INPUT
	XWRITEFILEEXECUTE : BOOL;
	XREADERRORFILEEXECUTE : BOOL;
	XENABLE : BOOL;
	INUMOFLISTELEMENTS : INT;
END_VAR
VAR_OUTPUT
	XWRITEFILEDONE : BOOL;
	XWRITEFILEBUSY : BOOL;
	XWRITEFILEERROR : BOOL;
	XERRORDETECTED : BOOL;
	XCHECKCONSISTENCYFAIL : BOOL;
	XDONE : BOOL;
	XBUSY : BOOL;
	AL_MC4P_LISTELEMENT : ARRAY [0..(ciArrayBreite + ciArrayHistory)] OF L_MC4P_ListElement;
	INUMOFLISTELEMENTSOUT : INT;
	APLISTELEM : ARRAY [0..(ciArrayBreite + ciArrayHistory)] OF POINTER TO L_MC4P_ListElement;
	ILISTHISTORYEND : INT := 1;
	ASCLISTHISTORY : ARRAY [1..ciArrayHistory] OF L_MC4P_ListElement;
END_VAR
VAR
	CIARRAYHISTORY : INT := 10;
	CIARRAYTIEFE : INT := 1000;
	CIARRAYBREITE : INT := 30;
	XTESTINMOTIONTASK : BOOL := FALSE;
	XFREETASKBUSY_INT : BOOL;
	XFREETASKDONE_INT : BOOL;
	XFREETASKERROR_INT : BOOL;
	EFREETASKEERRORID_INT : L_IE1P_Error;
	RES : SYSFILE.RTS_IEC_ResULT;
	HFILE : SYSFILE.RTS_IEC_HANDLE;
	XWFSIZE : __XWORD;
	XWRESULTWRITESTRING : __XWORD;
	FB_STACKDIAGDATA : L_MC1P_StackControlArray := STRUCT(iMaxLegth := ciArrayTiefe);
	ASCDIAGDATA : ARRAY [0..ciArrayTiefe] OF L_MC4P_PathListDiagnosticData;
	SCDIAGDATATMP : L_MC4P_PathListDiagnosticData;
	WSTEP : WORD := 0;
	WSTEPREF : WORD := 0;
	WSTEPWEF : WORD := 0;
	WSTEPWF : WORD := 0;
	XDATACHENGED : BOOL;
	XCONSISTENCY : BOOL;
	XWRITEFILEEXECUTE_OLD : BOOL;
	IDX : INT;
	INUMOFLISTELEMENTS_INT : INT;
	PLISTELEMENTLAST : POINTER TO L_MC4P_ListElement;
	PLISTELEMENTFIRST : POINTER TO L_MC4P_ListElement;
	PLEFT : POINTER TO L_MC4P_ListElement;
	OPEN2 : FILE.Open;
	CLOSE2 : FILE.Close;
	READ1 : FILE.Read;
	ASHEADLINE : ARRAY [1..10] OF STRING(255) := ['Hinweise zur ListenElementen:  Segmentnummer +2000:  Element aus Ipo,  Segmentnummer +1000:  diSegmentNoCopiedFrom $N', 'Hinweise zur Exeltabelle: oben ist der älteste und unten ist der akttuelste Stand der Liste  $N', 'Zeile1:AnzahlDurchläufe $TxPathStopExecute $TdiActFunID $TdiBusyFunID $TdiFunID $TlrOverride $T $TSegmente  $N', 'Zeile2: AbsZähler $TxPathStopExecute $TdiActFunID $TdiBusyFunID $TdiFunID, $TlrOverride $T $TMaske $T $N', '$N '];
	STABULATOR : STRING(2) := '$T';
	SLINEFEED : STRING(2) := '$N';
	SZEILE : STRING(255);
	SZEILE2 : STRING(255);
	IDATAIDX1 : INT;
	SEXELFILENAME : STRING;
	SLISTELEMENTFILENAME : STRING;
	SLISTELEMENTFILENAMEBASE : STRING;
	XREADERRORFILEDONE : BOOL;
	XREADERRORFILEBUSY : BOOL;
	XREADERRORFILEERROR : BOOL;
	XWRITEFILEEXECUTE_INTERN : BOOL;
	XREADERRORFILEEXECUTE_INTERN : BOOL;
	XREADERRORFILEEXECUTE_OLD : BOOL;
	DITIMESTAMP : DINT;
	ILISTHISTORYENDLENGTH : INT;
	SCLISTELEMENTEMPTY : L_MC4P_ListElement;
	IDX2 : INT;
	IDX3 : INT;
	ILISTELEMACTIVE : INT;
	IDATANO : INT;
	XAGERORR : BOOL;
	ASCAGEERRORINFO : ARRAY [0..7] OF L_IE1P_ErrorInformation;
	XSAVEAGERROR : BOOL;
	WLOOKAHEADHORIZON : WORD;
	DWTASKYCLE_US : DWORD;
	EACTIVEERRORID : L_IE1P_Error;
	SAXESGROUPNAME : STRING;
	XWRITEINMOTIONTASK : BOOL;
END_VAR
END_FUNCTION_BLOCK

METHOD CALL_CHECKCHANGES_SCDIAGDATA : BOOL
VAR_IN_OUT
	SCDIAGDATANEW : L_MC4P_PathListDiagnosticData;
	SCDIAGDATAOLD : L_MC4P_PathListDiagnosticData;
END_VAR
END_METHOD

METHOD CALL_CHECKCONSISTENCY : BOOL
VAR_IN_OUT
	SCDIAGDATA : L_MC4P_PathListDiagnosticData;
END_VAR
END_METHOD

METHOD CALL_INIT_SCDIAGDATA
VAR_IN_OUT
	SCDIAGDATA : L_MC4P_PathListDiagnosticData;
END_VAR
END_METHOD

METHOD CHECKCONSISTENCY
END_METHOD

METHOD READERRORFILE
END_METHOD

METHOD MAINFB : BOOL
VAR_INPUT
	PAXESGROUP : POINTER TO AXES_GROUP_KIN;
END_VAR
END_METHOD

METHOD CALL_WRITEEXELFILE
END_METHOD

METHOD CALL_WRITESEGEMENTFILE
VAR_IN_OUT
	SCLISTELEM : L_MC4P_ListElement;
END_VAR
END_METHOD

METHOD EXECUTEFREERUNTASK
END_METHOD

METHOD MAIN
END_METHOD

METHOD RESETREADDATA
END_METHOD

METHOD ABORT : UDINT
END_METHOD

METHOD EXECUTE : UDINT
END_METHOD

(* ---- L_MC4P_PATHREFFROMFILE.pou ---- *)
FUNCTION_BLOCK L_MC4P_PATHREFFROMFILE
VAR_INPUT
	XEXECUTE : BOOL;
	SFILENAME : STRING;
	XABORT : BOOL;
	DWSKIPMASK : DWORD := 0;
	LIBLOCKSEARCHLINENO : LINT := 0;
END_VAR
VAR_OUTPUT
	XDONE : BOOL;
	XBUSY : BOOL;
	XCOMMANDABORTED : BOOL;
	XERROR : BOOL;
	EERRORID : L_IE1P_Error;
	XDECODING : BOOL;
	LILINENODECODED : LINT;
	SLINEDECODED : STRING;
END_VAR
VAR
	LIBLOCKSEARCHLINENO_INT : LINT;
	IFILENO_INT : INT;
	XINTERPRETERHALT_INT : BOOL;
	XMOVEPATHACTIVE_INT : BOOL;
	WACTIVEMFUNCTION_INT : WORD;
	LISOURCELINENO_INT : LINT;
	XABORTACTIVE : BOOL;
	_XDONE : BOOL;
	_XBUSY : BOOL;
	_XCOMMANDABORTED : BOOL;
	_XDECODING : BOOL;
	SFILEADRESS : STRING;
	ITACKEDNUMOFELEMENTSINCYCLE_INT : INT := 0;
	IDECODEMAXNUMOFELEMENTS_INT : INT := 2;
	IDECODEMAXNUMOFELEMENTSFIRSTTIME_INT : INT := 3;
	IDECODENUMOFELEMENTS_INT : INT;
	FB_DECODENCPROGDATA : L_MC1P_StackControlArray := STRUCT(iMaxLegth := GVL_MovePath.gciNumOfPathFiles);
	SCHEADDATA : L_MC4P_AsciiDecoderHeadData;
	RSCACTFILEDATA : REFERENCE TO L_MC4P_AsciiDecoderFileData;
	XHALTATMOS_INT : BOOL := TRUE;
	XIGNOREMCOMMANDS_INT : BOOL;
	XNEWFILE_INT : BOOL;
	LRCIRCLTARGETTOLERANCE_INT : LREAL := 0.1;
	FB_SEMA : L_MC1P_CriticalSection;
	ITAKEELEMENTCNT : INT;
	IADDELEMENTCNT : INT;
	FB_DECODEMOVEDATALOWTASK : L_MC1P_StackControlArray := STRUCT(iMaxLegth := GVL_MovePath.gciNumOfDecodeAsciiData);
	FB_DECODEMOVEDATAMOTIONTASK : L_MC1P_StackControlArray := STRUCT(iMaxLegth := GVL_MovePath.gciNumOfDecodeAsciiData);
	ASCDECODEMOVEDATA_INT : ARRAY [1..GVL_MovePath.gciNumOfDecodeAsciiData] OF L_MC4P_Parameter_MCMove;
	IELEMENINARRAYDECODING : INT;
	FB_DECODEMOVEDATALOWTASK_RESERVE : L_MC1P_StackControlArray := STRUCT(iMaxLegth := GVL_MovePath.gciNumOfDecodeAsciiData_reserve);
	ASCDECODEMOVEDATA_RESERVE : ARRAY [1..GVL_MovePath.gciNumOfDecodeAsciiData_reserve] OF L_MC4P_Parameter_MCMove;
	XERROR_DECODERENDLOOP : BOOL;
	DWTIMEOUTCNT : DWORD := 0;
	DWTIMEOUT : DWORD := 100000;
	XERROR_TIMEOUT : BOOL;
	DWTIMEOUT_MASK : DWORD;
	WTIMEOUTDECODERSTATE : WORD;
	WSTATE : WORD;
	XID1 : BOOL;
	XWID_INT : POINTER TO BOOL := ADR(xId1);
	XSETPATHDATAACTIVE_INT : BOOL;
	XSETPATHDATAACTIVE_OLD : BOOL;
	REQUESTSINFO : DWORD;
	REQUESTSINFO_OLD : DWORD;
	DWRTRIG : DWORD;
	DWFTRIG : DWORD;
	XRESETOUTPUTS : BOOL;
	XERROR_INVALIDSYNCDATA : BOOL;
	BYERRORADRESS : BYTE;
	STERRORADRESSVALUE : STRING;
	XPATHREFABORT : BOOL;
	XDECODEINNEXTTASKCYCLE : BOOL;
	XFBISABORTED : BOOL;
	SFILE_INT : STRING := '';
	XDECODEBUSY_INT : BOOL;
	XDECODEDONE_INT : BOOL;
	XDECODEERROR_INT : BOOL;
	EDECODEEERRORID_INT : L_IE1P_Error;
	DWINTERNALID_INT : DWORD;
	STDECODEERRORLINE : STRING;
	RES : SYSFILE.RTS_IEC_RESULT;
	HFILE : SYSFILE.RTS_IEC_HANDLE;
	UDILENGTHFILE : UDINT;
	XTESTINMOTIONTASK : BOOL := FALSE;
	EXCEPTIONCODE : __SYSTEM.ExceptionCode;
	DWPREDECODERIDLECYCLES : DWORD := 0;
	DWPOSTDECODERIDLECYCLES : DWORD := 0;
	BLOCKSEARCHENABLED : BOOL;
	DATATYPE : WORD;
	DWTIMEOUTMASK : DWORD;
	ENDELEMENT : POINTER TO L_MC4P_Parameter_MCMove;
	ENDIDX : INT;
	POSTDECODERIDLECYCLES : DWORD;
	PREDECODERIDLECYCLES : DWORD;
	SETCIRCTARGETTOLERANCE : LREAL;
	SIZE : UDINT;
	STARTELEMENT : POINTER TO L_MC4P_Parameter_MCMove;
	STARTIDX : INT;
	STERRORCOMMAND : STRING;
	TAKEELEMENT : POINTER TO L_MC4P_Parameter_MCMove;
	XDECODEINMOTIONTASK : BOOL;
	XHALTATMOS : BOOL;
	XIGNOREMCOMMANDS : BOOL;
	XINTERPRETERHALT : BOOL;
END_VAR
END_FUNCTION_BLOCK

METHOD ABORTFB
END_METHOD

METHOD CALL_ALLOCPOINTADR
END_METHOD

METHOD CALL_ERRORHANDLER
END_METHOD

METHOD CALL_FBMETHODS
END_METHOD

METHOD CALL_OUTPUT
END_METHOD

METHOD CALL_REQUESTS_EXT
END_METHOD

METHOD CALL_RESETCOMMANDS
END_METHOD

METHOD CALL_RESETOUTPUT
END_METHOD

METHOD CALL_RESETSTATUS
END_METHOD

METHOD CALL_STATEMACHINE
END_METHOD

METHOD CALL_SYNCDECODEMOVEDATA
END_METHOD

METHOD FUN_DECODEAUX : BOOL
VAR_IN_OUT
	STADRESSVALUE : STRING(255);
	SCDECODEHEADDATA : L_MC4P_AsciiDecoderHeadData;
END_VAR
END_METHOD

METHOD FUN_DECODEADRESS : BOOL
VAR_OUTPUT
	XERROR : BOOL;
	EERRORID : L_IE1P_Error;
END_VAR
VAR_IN_OUT
	BYADRESS : BYTE;
	STADRESSVALUE : STRING(255);
	SCDECODEHEADDATA : L_MC4P_AsciiDecoderHeadData;
END_VAR
END_METHOD

METHOD FUN_DECODEG : BOOL
VAR_IN_OUT
	LIADRESSVALUE : LINT;
	SCDECODEHEADDATA : L_MC4P_AsciiDecoderHeadData;
END_VAR
END_METHOD

METHOD FUN_DECODEGOTO : BOOL
VAR_OUTPUT
	XERROR : BOOL;
	EERRORID : L_IE1P_Error;
END_VAR
VAR_IN_OUT
	STADRESSVALUE : STRING(255);
	SCDECODEHEADDATA : L_MC4P_AsciiDecoderHeadData;
END_VAR
END_METHOD

METHOD FUN_DECODEH : BOOL
VAR_IN_OUT
	STADRESSVALUE : STRING(255);
	SCDECODEHEADDATA : L_MC4P_AsciiDecoderHeadData;
	XERROR : BOOL;
	EERRORID : L_IE1P_Error;
END_VAR
END_METHOD

METHOD FUN_DECODEI : BOOL
VAR_IN_OUT
	STADRESSVALUE : STRING(255);
	SCDECODEHEADDATA : L_MC4P_AsciiDecoderHeadData;
END_VAR
END_METHOD

METHOD FUN_DECODEIFCASE : BOOL
VAR_INPUT
	STLINE : STRING(255);
END_VAR
VAR_OUTPUT
	XERROR : BOOL;
	EERRORID : L_IE1P_Error;
END_VAR
VAR_IN_OUT
	SCDECODEHEADDATA : L_MC4P_AsciiDecoderHeadData;
END_VAR
END_METHOD

METHOD FUN_DECODEL : BOOL
VAR_IN_OUT
	STADRESSVALUE : STRING(255);
	SCDECODEHEADDATA : L_MC4P_AsciiDecoderHeadData;
	XERROR : BOOL;
	EERRORID : L_IE1P_Error;
END_VAR
END_METHOD

METHOD FUN_DECODELINE : BOOL
VAR_OUTPUT
	XGETNEXTSOURCELINE : BOOL;
	XELEMENTDECODED : BOOL;
	XERROR : BOOL;
	EERRORID : L_IE1P_Error;
END_VAR
VAR_IN_OUT
	SCDECODEHEADDATA : L_MC4P_AsciiDecoderHeadData;
	SCDECODEMOVEDATA : L_MC4P_Parameter_MCMove;
END_VAR
END_METHOD

METHOD FUN_DECODEM : BOOL
VAR_IN_OUT
	LIADRESSVALUE : LINT;
	SCDECODEHEADDATA : L_MC4P_AsciiDecoderHeadData;
	XERROR : BOOL;
	EERRORID : L_IE1P_Error;
END_VAR
END_METHOD

METHOD FUN_DECODEN : BOOL
VAR_IN_OUT
	STADRESSVALUE : STRING(255);
	SCDECODEHEADDATA : L_MC4P_AsciiDecoderHeadData;
END_VAR
END_METHOD

METHOD FUN_DECODEO : BOOL
VAR_IN_OUT
	STADRESSVALUE : STRING(255);
	SCDECODEHEADDATA : L_MC4P_AsciiDecoderHeadData;
	XERROR : BOOL;
	EERRORID : L_IE1P_Error;
END_VAR
END_METHOD

METHOD FUN_DECODEP : BOOL
VAR_IN_OUT
	STADRESSVALUE : STRING(255);
	SCDECODEHEADDATA : L_MC4P_AsciiDecoderHeadData;
END_VAR
END_METHOD

METHOD FUN_DELETECOMMENTS : BOOL
VAR_OUTPUT
	STCOMMENT : STRING;
	ILINESIZE : INT;
END_VAR
VAR_IN_OUT
	STLINE : STRING(255);
END_VAR
END_METHOD

METHOD FUN_DELETECOMMENTS_TYPE1 : BOOL
VAR_IN_OUT
	STLINE : STRING(255);
	STCOMMENT : STRING;
	ICOMMENTPOS : INT;
END_VAR
END_METHOD

METHOD FUN_DELETECOMMENTS_TYPE2 : BOOL
VAR_INPUT
	ICOMMENTTYPE : INT;
END_VAR
VAR_IN_OUT
	STLINE : STRING(255);
	STCOMMENT : STRING;
END_VAR
END_METHOD

METHOD FUN_FINDJUMPTARB : BOOL
VAR_INPUT
	LIJUMPTARGET : LINT;
	UDIFILELENGTH : UDINT;
	UDIPOS : UDINT;
	UDIPOSSTART : UDINT;
END_VAR
VAR_OUTPUT
	UDITARLINEPOS : UDINT;
	XERROR : BOOL;
	EERRORID : L_IE1P_Error;
END_VAR
END_METHOD

METHOD FUN_FINDJUMPTARF : BOOL
VAR_INPUT
	LIJUMPTARGET : LINT;
	UDIFILELENGTH : UDINT;
	UDIPOS : UDINT;
END_VAR
VAR_OUTPUT
	UDITARLINEPOS : UDINT;
	XERROR : BOOL;
	EERRORID : L_IE1P_Error;
END_VAR
END_METHOD

METHOD FUN_GOTO : BOOL
VAR_OUTPUT
	XERROR : BOOL;
	EERRORID : L_IE1P_Error;
END_VAR
VAR_IN_OUT
	SCDECODEHEADDATA : L_MC4P_AsciiDecoderHeadData;
	STLINE : STRING(255);
END_VAR
END_METHOD

METHOD FUN_GETADRESS : BOOL
VAR_OUTPUT
	ILINESIZE : INT;
	BYADRESS : BYTE;
	SADRESSVALUE : STRING;
END_VAR
VAR_IN_OUT
	STLINE : STRING(255);
END_VAR
END_METHOD

METHOD FUN_ISALPHACHAR : BOOL
VAR_INPUT
	BYCHAR : BYTE;
END_VAR
END_METHOD

METHOD FUN_READLINE : L_IE1P_Error
VAR_INPUT
	UDIPOSIN : UDINT;
	XEXITCLOSEFILE : BOOL;
	XFINDSTARTCOMAND : BOOL;
END_VAR
VAR_OUTPUT
	UDIPOSOUT : UDINT;
	ILINESIZE : INT;
	IPOSLF : INT;
	IPOSNL : INT;
	UDIRESULTFILEOPEN : UDINT;
	UDIRESULTREADSTRING : UDINT;
	XENDOFFILE : BOOL;
	XLASTLINE : BOOL;
	XSTART : BOOL;
END_VAR
VAR_IN_OUT
	HFILE : SYSFILE.RTS_IEC_HANDLE;
	RES : SYSFILE.RTS_IEC_ResULT;
	STLINE : STRING(255);
END_VAR
END_METHOD

METHOD FUN_READLINEBACK : BOOL
VAR_INPUT
	UDIPOSIN : UDINT;
	XEXITCLOSEFILE : BOOL;
	UDIPOSSTART : UDINT := 0;
END_VAR
VAR_OUTPUT
	UDIPOSOUT : UDINT;
	ILINESIZE : INT;
	UDIRESULTFILEOPEN : UDINT;
	XSTARTOFFILE : BOOL;
END_VAR
VAR_IN_OUT
	HFILE : SYSFILE.RTS_IEC_HANDLE;
	RES : SYSFILE.RTS_IEC_ResULT;
	STLINE : STRING(255);
END_VAR
END_METHOD

METHOD FUN_REPLACEVAR : BOOL
VAR_IN_OUT
	STVALUE : STRING(255);
END_VAR
END_METHOD

METHOD FUN_STRING_PLCVARIABLE_TO_LINT : BOOL
VAR_INPUT
	STVALUE : STRING(255);
END_VAR
VAR_OUTPUT
	LIVALUE : LINT;
END_VAR
END_METHOD

METHOD FUN_STRING_PLCVARIABLE_TO_LREAL : BOOL
VAR_INPUT
	STVALUE : STRING(255);
END_VAR
VAR_OUTPUT
	LRVALUE : LREAL;
END_VAR
END_METHOD

METHOD FUN_STRING_TO_LINT : BOOL
VAR_INPUT
	STVALUE : STRING;
	XVARALLOWED : BOOL;
END_VAR
VAR_OUTPUT
	LIVALUE : LINT;
END_VAR
END_METHOD

METHOD FUN_STRING_TO_LREAL : BOOL
VAR_INPUT
	STVALUE : STRING(255);
END_VAR
VAR_OUTPUT
	LRVALUE : LREAL;
END_VAR
END_METHOD

METHOD FUN_SHUNTINGYARD : BOOL
VAR_INPUT
	STVALUE : STRING(255);
END_VAR
VAR_OUTPUT
	SCVALUE : L_UBUP_Variable;
END_VAR
END_METHOD

METHOD CALL_DECODER
END_METHOD

METHOD CALL_DECODER_READASCIIFILE
END_METHOD

METHOD EXECUTEFREERUNTASK
END_METHOD

METHOD FUN_CLOSEFILE
END_METHOD

METHOD INIT_HEADDATA
VAR_IN_OUT
	SCDECODEHEADDATA : L_MC4P_AsciiDecoderHeadData;
END_VAR
END_METHOD

METHOD MAIN
END_METHOD

METHOD GETID : __XWORD
END_METHOD

METHOD GETPATHDATA : ARRAY [1..GVL_MovePath.gciNumOfDecodeAsciiData] OF POINTER TO L_MC4P_Parameter_MCMove
END_METHOD

METHOD GETPATHDATAACTIVE : BOOL
END_METHOD

METHOD GETSTATUS : DWORD
END_METHOD

METHOD SETABORT
END_METHOD

METHOD SETACTIVEMFUNCTION
VAR_INPUT
	WACTIVEMFUNCTION : WORD;
END_VAR
END_METHOD

METHOD SETMOVEPATHACTIVE
VAR_INPUT
	XMOVEPATHACTIVE : BOOL;
END_VAR
END_METHOD

METHOD SETPATHDATAACTIVE
VAR_INPUT
	XPATHDATAACTIVE : BOOL;
END_VAR
END_METHOD

METHOD CALL_INIT
END_METHOD

METHOD CALL_S000_CYCLIC
END_METHOD

METHOD ABORT : UDINT
END_METHOD

METHOD EXECUTE : UDINT
END_METHOD

(* ---- L_MC4P_PATHREFMONITOR.pou ---- *)
FUNCTION_BLOCK L_MC4P_PATHREFMONITOR
VAR_INPUT
	XEXECUTE : BOOL;
	XABORT : BOOL;
	ITFPATHREF : MC_PATH_REF;
	SCSKIP : L_MC4P_SkipGCode;
	ASCDATA : POINTER TO L_MC4P_PathRefMonitorData;
END_VAR
VAR_OUTPUT
	XDONE : BOOL;
	XBUSY : BOOL;
	XCOMMANDABORTED : BOOL;
	XERROR : BOOL;
	EERRORID : L_IE1P_Error;
	UDINEWESTELEMENT : UDINT;
	UDIELEMENTCOUNT : UDINT;
END_VAR
VAR
	_ITFPATHREF : MC_PATH_REF;
	_UDISTARTIDX : UDINT;
	_UDIENDIDX : UDINT;
	_UDIREADIDX : UDINT;
	_UDILOWER : UDINT;
	_UDIUPPER : UDINT;
	_UDISIZE : UDINT;
	_DWSTATUS : DWORD;
	_XREINIT : BOOL := FALSE;
	_XDATADIALOG : BOOL := FALSE;
	_UDIVISUARRIDX : UDINT := 0;
	_PSCDATAARR : POINTER TO L_MC4P_PathRefMonitorData;
	_PSCDATAVISU : POINTER TO L_MC4P_PathRefMonitorData;
	_SCDATAINITIAL : L_MC4P_PathRefMonitorData;
	_ISKIPVIEWFRAME : INT := 0;
	_MODEL : L_UBUP_BehaviourModel_ETrigA;
END_VAR
END_FUNCTION_BLOCK

METHOD MAPOUTPUTS
END_METHOD

METHOD CYCLICACTION
VAR_INPUT
	ITFTIMINGCONTROLLER : L_UBUP.L_UBUP_ITimingController;
END_VAR
VAR_OUTPUT
	XCOMPLETE : BOOL;
	XABORT : BOOL;
	IERRORID : INT;
END_VAR
END_METHOD

METHOD FINALIZEACTION
VAR_INPUT
	XABORTPROPOSED : BOOL;
	IERRORIDPROPOSED : INT;
END_VAR
VAR_OUTPUT
	XCOMPLETE : BOOL;
	XABORT : BOOL;
	IERRORID : INT;
END_VAR
END_METHOD

METHOD RESETACTION
VAR_OUTPUT
	XCOMPLETE : BOOL;
END_VAR
END_METHOD

METHOD STARTACTION
VAR_OUTPUT
	XCOMPLETE : BOOL;
	IERRORID : INT;
END_VAR
END_METHOD

METHOD FB_INIT : BOOL
VAR_INPUT
	BINITRETAINS : BOOL;
	BINCOPYCODE : BOOL;
END_VAR
END_METHOD

METHOD APPENDDATASET : BOOL
VAR_INPUT
	PMCMOVE : POINTER TO L_MC4P_Parameter_MCMove;
END_VAR
END_METHOD

METHOD SKIP : BOOL
VAR_INPUT
	PMCMOVE : POINTER TO L_MC4P_Parameter_MCMove;
END_VAR
END_METHOD

(* ---- L_MC4P_PICKANDPLACEMEMORY.pou ---- *)
FUNCTION_BLOCK L_MC4P_PICKANDPLACEMEMORY
VAR_INPUT
	FB_SEMAMOVEFBS : L_MC1P_CriticalSection;
	AMC_MOVELINREL : ARRAY [1..3] OF L_MC4P_MoveLinearRelative_Internal;
	AFB_MOVEELLIPTICAL : ARRAY [1..3] OF L_MC4P_MoveEllipticalAbsolutePnP_Internal;
	AFB_MOVESPLINE : ARRAY [1..3] OF L_MC4P_MoveSplinePnP_Internal;
	AMC_MOVELINABS1 : ARRAY [1..10] OF L_MC4P_MoveLinearAbsolute_Internal;
	AMC_MOVELINABS2 : ARRAY [1..10] OF L_MC4P_MoveLinearAbsolute_Internal;
	AMC_MOVELINABS3 : ARRAY [1..10] OF L_MC4P_MoveLinearAbsolute_Internal;
	AMC_MOVELINABS4 : ARRAY [1..3] OF L_MC4P_MoveLinearAbsolute_Internal;
	AMC_MOVELINABS5 : ARRAY [1..2] OF L_MC4P_MoveLinearAbsolute_Internal;
	AMC_MOVEDIRABS1 : ARRAY [1..10] OF L_MC4P_MoveDirectAbsolute_Internal;
	AMC_MOVEDIRABS2 : ARRAY [1..10] OF L_MC4P_MoveDirectAbsolute_Internal;
	AMC_MOVEDIRREL : ARRAY [1..1] OF L_MC4P_MoveDirectRelative_Internal;
	AFB_GROUPWAITTIME : ARRAY [1..3] OF L_MC4P_GroupWaitTime_Internal;
	ASCPROFILEPARMEM : ARRAY [1..10] OF ARRAY [1..10] OF L_MC4P_scPickAndPlaceProfileParState;
	ASCPROFILETIMEFROMCVTARGET : ARRAY [1..16] OF ARRAY [0..10] OF L_MC4P_MeasuredProfileTime;
	AIRINGMEMPROFILETIME : ARRAY [1..16] OF ARRAY [1..2] OF INT;
	FB_SEMA : L_MC1P_CriticalSection;
	CONVEYORBELTVIRTUAL : ARRAY [1..2] OF AXIS_REF := [STRUCT(UsedAsInternalAxisInstance := TRUE), STRUCT(UsedAsInternalAxisInstance := TRUE)];
END_VAR
END_FUNCTION_BLOCK

(* ---- L_MC4P_PREPAREPATH.pou ---- *)
FUNCTION_BLOCK L_MC4P_PREPAREPATH EXTENDS L_MC4P_Template_KIN
VAR_INPUT
	PLIST : POINTER TO L_MC4P_PathDataList;
	PPATHELEMENT : POINTER TO L_MC4P_PathElement;
	ALRSTARTPOS : ARRAY [1..12] OF LREAL;
	PAXESGROUP : POINTER TO AXES_GROUP_KIN;
	XINITSTATEMACHINE : BOOL;
	PCORRESPONDINGFB : POINTER TO L_MC4P_MoveContPath;
	XCHECKWORKSPACE : BOOL := TRUE;
	UDICHECKWORKSPACESTEPS : UDINT := 5;
END_VAR
VAR_OUTPUT
	XERROR : BOOL := FALSE;
	ERRORID : L_IE1P_Error;
	DWINTERNALERRORID : DWORD;
END_VAR
VAR
	SCERROR : L_MC4P_ErrorStruct;
	XNOBLENDINGERRORS : BOOL := TRUE;
	XDOPREPARE : BOOL := FALSE;
	PLISTELEMENT : POINTER TO L_MC4P_ListElement;
	PLISTELEMENT_PREVIOUS : POINTER TO L_MC4P_ListElement;
	PLISTELEMENTSTART : POINTER TO L_MC4P_ListElement;
	PLISTELEMENTEND : POINTER TO L_MC4P_ListElement;
	PLISTELEMENT_IDENTPTPTYPE : POINTER TO L_MC4P_ListElement;
	PLISTELEMENT_CALCPTPPROFILE : POINTER TO L_MC4P_ListElement;
	WSTEP : WORD := 0;
	PTP_PREPSTATE : L_MC4P_PTPPrepStates;
	BIDENTTMAX_INIT : BOOL;
	BIDENTPTPTYPE_INIT : BOOL;
	BCALCPTPPROFILE_INIT : BOOL;
	ACHSE : UINT;
	CNTCYCLESPREPAREPATH : UINT;
	CNTCYCLESPREPAREPATHMAX : UINT := 500;
	BYAUXAXISSEQCOUNT : BYTE;
	PLISTELEMENTAUXSEQSTART : ARRAY [1..6] OF POINTER TO L_MC4P_ListElement;
	PLISTELEMENTAUXSEQEND : ARRAY [1..6] OF POINTER TO L_MC4P_ListElement;
	XRECALCPROFILES : BOOL;
	XAUXAXISACTIVNEWSET : BOOL;
	PTESTAUX : POINTER TO L_MC4P_ListElement;
	XFOUND : BOOL;
	LRTIMEELEMENT : LREAL;
	LRJERKDEC : LREAL;
	DWIPOSTATE : DWORD;
	LRTIMELIST : LREAL;
	LRTIMEIPO : LREAL;
	LRTIMEREST : LREAL;
	LRTIMETOCUT : LREAL;
	LRTIMEACCZERO : LREAL;
	LRSTARTACC : LREAL;
	LRSTARTVEL : LREAL;
	LRSTARTPOS : LREAL;
	LRENDACC : LREAL;
	LRENDVEL : LREAL;
	LRENDPOS : LREAL;
	DWBOTHDIRECTIONS : DWORD := 3;
	SCPROFILEPARAMETER : L_MC1P_ProfileParameter;
	SCPROFILEDATA : L_MC1P_ProfileData;
	PLISTELEMENTTMP : POINTER TO L_MC4P_ListElement;
	WCPP_ABC_STEP : WORD;
	WCPPSTEP : WORD;
	LRVIN_ORIGINAL : LREAL;
	LRVOUT_ORIGINAL : LREAL;
	XDOPROFILECHECK : BOOL := FALSE;
	WDOPREPARECOUNTER : WORD;
	WDOPREPARECOUNTERMAX : WORD := 1;
	WLDE_MODE : WORD := 2;
	LRANGULARTOLERANCE_LDC : LREAL := 0.1;
	LRMAXACCDIFF_LDC : LREAL := 0.0;
	LRACCREDFACTOR : LREAL := 0.1;
	TIMESTART : ULINT;
	TIMEEND : ULINT;
	AXTAKETIMESTAMP : ARRAY [0..20] OF BOOL;
	ULIPREPPATHTIME : ARRAY [0..20] OF ULINT;
	DWSCHELLINGWORKAROUNDCOUNTER : DWORD := 0;
	DIRESETBLENDINGSEGMENTNO : DINT := 0;
	DIBLENDINGSEGMENTNORESETTED : DINT := 0;
	XBLENDINGALWAYSSHORTESTWAY : BOOL := FALSE;
	XENABLECORRLDS00042356 : BOOL := TRUE;
	SCSP : L_MC4P_CyclicData;
	LRPERCLENGTHDELTA : LREAL := 0.1;
	LRFACTOR : LREAL := (1 / (1.0 - (0.1 * lrPercLengthDelta)));
END_VAR
END_FUNCTION_BLOCK

METHOD ACTIVATESEGMENT
VAR_INPUT
	PLISTELEMENT : POINTER TO L_MC4P_ListElement;
END_VAR
END_METHOD

METHOD AUXAXISCALCMAINPATHLENGTH : BOOL
VAR_INPUT
	PLISTELEMENT : POINTER TO L_MC4P_ListElement;
	IDX : INT;
END_VAR
VAR_OUTPUT
	LRMAINAXPATH : LREAL;
	PLISTELEMENTAUXSEQSTART : POINTER TO L_MC4P_ListElement;
END_VAR
END_METHOD

METHOD AUXAXISCALCMAINTIME : BOOL
VAR_INPUT
	PLISTELEMENT : POINTER TO L_MC4P_ListElement;
	IDX : INT;
END_VAR
VAR_OUTPUT
	LRMAINTIMECOMPLETE : LREAL;
	LRMAINAXPATH : LREAL;
	PLISTELEMENTAUXSEQSTART : POINTER TO L_MC4P_ListElement;
END_VAR
END_METHOD

METHOD AUXAXISLIMITMAINAXIS
VAR_INPUT
	PLISTELEMENT : POINTER TO L_MC4P_ListElement;
END_VAR
VAR_OUTPUT
	XRECALCPROFILES : BOOL := FALSE;
END_VAR
END_METHOD

METHOD AUXAXISPREPARE
VAR_INPUT
	PLISTELEMENT : POINTER TO L_MC4P_ListElement;
END_VAR
VAR_OUTPUT
	XRECALCPROFILES : BOOL := FALSE;
END_VAR
END_METHOD

METHOD CALCULATEORIPATH
VAR_INPUT
	PLISTELEMENTDATA : POINTER TO L_MC4P_ListElementData;
END_VAR
END_METHOD

METHOD CALCULATEPTPTARGET
VAR_INPUT
	PLISTELEMENTDATA : POINTER TO L_MC4P_ListElementData;
END_VAR
END_METHOD

METHOD CALCULATEPATHPOLYNOM
VAR_INPUT
	PLISTELEMENT : POINTER TO L_MC4P_ListElement;
END_VAR
END_METHOD

METHOD CALCULATEPROFILEABC
VAR_INPUT
	PLISTELEMENT : POINTER TO L_MC4P_ListElement;
END_VAR
VAR_OUTPUT
	XSTEPBACK : BOOL;
END_VAR
END_METHOD

METHOD CALCULATEPROFILEPOLYNOM
VAR_INPUT
	PLISTELEMENT : POINTER TO L_MC4P_ListElement;
END_VAR
END_METHOD

METHOD CREATERESETBLENDINGLOG
END_METHOD

METHOD DETERMINEBLENDINGDIRECTION : BOOL
VAR_INPUT
	PREVIOUS : POINTER TO L_MC4P_ListElementData;
	BLENDING : POINTER TO L_MC4P_ListElementData;
	NEXT : POINTER TO L_MC4P_ListElementData;
END_VAR
END_METHOD

METHOD INTERPRETER
VAR_INPUT
	PPATHELEMENT : POINTER TO L_MC4P_PathElement;
END_VAR
VAR_IN_OUT
	PLIST : POINTER TO L_MC4P_PathDataList;
END_VAR
END_METHOD

METHOD LIMITDYNAMICSCOMBINE
VAR_INPUT
	PLISTELEMENT : POINTER TO L_MC4P_ListElement;
END_VAR
END_METHOD

METHOD LIMITDYNAMICSCORNER
VAR_INPUT
	PLISTELEMENT : POINTER TO L_MC4P_ListElement;
END_VAR
END_METHOD

METHOD LIMITDYNAMICSELEMENTS
VAR_INPUT
	PLISTELEMENT : POINTER TO L_MC4P_ListElement;
END_VAR
END_METHOD

METHOD LIMITDYNAMICSPATHLENGTH
VAR_INPUT
	PLISTELEMENTSTART : POINTER TO L_MC4P_ListElement;
	PLISTELEMENTEND : POINTER TO L_MC4P_ListElement;
END_VAR
END_METHOD

METHOD LIMITDYNAMICSPATHLENGTH_KART
VAR_INPUT
	PLISTELEMENTSTART : POINTER TO L_MC4P_ListElement;
	PLISTELEMENTEND : POINTER TO L_MC4P_ListElement;
END_VAR
END_METHOD

METHOD PREPAREPTPPROFILES
VAR_INPUT
	PLISTELEMENTSTART : POINTER TO L_MC4P_ListElement;
	PLISTELEMENTEND : POINTER TO L_MC4P_ListElement;
END_VAR
END_METHOD

METHOD PREPAREPTPPROFILES_CALCPTPPROFILE
VAR_INPUT
	PLISTELEMENTSTART : POINTER TO L_MC4P_ListElement;
	PLISTELEMENTEND : POINTER TO L_MC4P_ListElement;
END_VAR
VAR_OUTPUT
	XRETURN : BOOL;
END_VAR
END_METHOD

METHOD PREPAREPTPPROFILES_IDENTPTPTYPE
VAR_INPUT
	PLISTELEMENTSTART : POINTER TO L_MC4P_ListElement;
	PLISTELEMENTEND : POINTER TO L_MC4P_ListElement;
END_VAR
VAR_OUTPUT
	XRETURN : BOOL;
END_VAR
END_METHOD

METHOD PREPAREPTPPROFILES_IDENTTMAX
VAR_INPUT
	PLISTELEMENTSTART : POINTER TO L_MC4P_ListElement;
	PLISTELEMENTEND : POINTER TO L_MC4P_ListElement;
END_VAR
VAR_OUTPUT
	XRETURN : BOOL;
END_VAR
END_METHOD

METHOD PREPAREPTPPROFILES_QUITPREP
VAR_INPUT
	PLISTELEMENTSTART : POINTER TO L_MC4P_ListElement;
	PLISTELEMENTEND : POINTER TO L_MC4P_ListElement;
END_VAR
END_METHOD

METHOD RAISESWLIMITERROR : L_IE1P_Error
VAR_INPUT
	PLISTELEMENT : POINTER TO L_MC4P_ListElement;
	IDX : DINT;
END_VAR
END_METHOD

METHOD RESETPATHANDRESTART
END_METHOD

METHOD RESETPATHPREPARATION
END_METHOD

METHOD SMOOTHPATH
VAR_INPUT
	PLISTELEMENT : POINTER TO L_MC4P_ListElement;
END_VAR
END_METHOD

METHOD STRETCHPROFILETOTIME
VAR_INPUT
	PROFILEDATA_ACT : L_MC1P_ProfileData;
	PARAM_ACT : L_MC1P_ProfileParameter;
	T_DESIRED : LREAL;
END_VAR
VAR_OUTPUT
	PROFILEDATA_NEW : L_MC1P_ProfileData;
	PARAM_NEW : L_MC1P_ProfileParameter;
END_VAR
END_METHOD

METHOD CALC_RAST2VEL_TRAPONLY
VAR_INPUT
	POS_IN : LREAL;
	POS_OUT : LREAL;
	JERK : LREAL;
	AMAX : LREAL;
	T_DESIRED : LREAL;
END_VAR
VAR_IN_OUT
	SCPROFILEDATA : L_MC1P_ProfileData;
END_VAR
END_METHOD

METHOD CALC_RAST2VEL_TRIONLY
VAR_INPUT
	POS_IN : LREAL;
	POS_OUT : LREAL;
	JERK : LREAL;
	T_DESIRED : LREAL;
END_VAR
VAR_IN_OUT
	SCPROFILEDATA : L_MC1P_ProfileData;
END_VAR
END_METHOD

METHOD CALC_REDVMAX
VAR_INPUT
	ACT : POINTER TO L_MC4P_ListElementData;
	ACHSE : UINT;
	T_MAX_ACT : LREAL;
END_VAR
END_METHOD

METHOD CALC_VEL2RAST_TRAPONLY
VAR_INPUT
	POS_IN : LREAL;
	POS_OUT : LREAL;
	JERK : LREAL;
	V_IN : LREAL;
	AMAX : LREAL;
	T_DESIRED : LREAL;
END_VAR
VAR_IN_OUT
	SCPROFILEDATA : L_MC1P_ProfileData;
END_VAR
END_METHOD

METHOD CALC_VEL2RAST_TRIONLY
VAR_INPUT
	POS_IN : LREAL;
	POS_OUT : LREAL;
	JERK : LREAL;
	V_IN : LREAL;
	V_OUT : LREAL;
	AMAX : LREAL;
	T_DESIRED : LREAL;
END_VAR
VAR_IN_OUT
	SCPROFILEDATA : L_MC1P_ProfileData;
END_VAR
END_METHOD

METHOD CREATEABCELEMENTS
VAR_INPUT
	PLISTELEMENTCUT : POINTER TO L_MC4P_ListElement;
END_VAR
VAR_OUTPUT
	PLISTELEMENTCUT_1A : POINTER TO L_MC4P_ListElement;
	PLISTELEMENTCUT_1B : POINTER TO L_MC4P_ListElement;
	PLISTELEMENTCUT_1C : POINTER TO L_MC4P_ListElement;
	PLISTELEMENTCUT_2B : POINTER TO L_MC4P_ListElement;
	PLISTELEMENTCUT_2C : POINTER TO L_MC4P_ListElement;
	PNEW : POINTER TO L_MC4P_ListElement;
	PLEFT : POINTER TO L_MC4P_ListElement;
END_VAR
END_METHOD

METHOD IDENTCUTELEMENT
VAR_IN_OUT
	PLISTELEMENTCUT : POINTER TO L_MC4P_ListElement;
END_VAR
END_METHOD

METHOD LOOKAHEAD_CLEANUP
END_METHOD

METHOD LOOKAHEAD_PREPARE
END_METHOD

METHOD MODIFYABCELEMENTS
VAR_INPUT
	PLISTELEMENTCUT : POINTER TO L_MC4P_ListElement;
END_VAR
VAR_IN_OUT
	PLISTELEMENTCUT_1A : POINTER TO L_MC4P_ListElement;
	PLISTELEMENTCUT_1B : POINTER TO L_MC4P_ListElement;
	PLISTELEMENTCUT_1C : POINTER TO L_MC4P_ListElement;
END_VAR
END_METHOD

METHOD CALCMAXVELOUT : LREAL
VAR_INPUT
	LRJERK : LREAL;
	LRAMAX : LREAL;
	LRDIST : LREAL;
	LRVIN : LREAL;
END_VAR
END_METHOD

METHOD INITGEOOBJECT
VAR_INPUT
	PLISTELEMENT : POINTER TO L_MC4P_ListElement;
END_VAR
VAR_OUTPUT
	SCERROR : L_MC4P_ErrorStruct;
END_VAR
END_METHOD

METHOD CHECKWORKSPACE
VAR_INPUT
	PLISTELEMENT : POINTER TO L_MC4P_ListElement;
END_VAR
END_METHOD

METHOD CHECKWORKSPACEDOT
VAR_INPUT
	PLISTELEMENT : POINTER TO L_MC4P_ListElement;
	LRPERCLENGTH : LREAL;
	LRLENGTH : LREAL;
	SCTRAFOINFO_SW : REFERENCE TO L_MC4P_TrafoInfo;
	SCERROR : REFERENCE TO L_MC4P_ErrorStruct;
END_VAR
END_METHOD

(* ---- L_MC4P_READBOOLPARAMETER.pou ---- *)
FUNCTION_BLOCK L_MC4P_READBOOLPARAMETER EXTENDS L_MC4P_Template_AG_KIN
VAR_INPUT
	XENABLE : BOOL;
	DIPARAMETERNUMBER : DINT;
END_VAR
VAR_OUTPUT
	XVALID : BOOL;
	XBUSY : BOOL;
	XERROR : BOOL;
	EERRORID : L_IE1P_Error;
	XVALUE : BOOL;
END_VAR
VAR
	XENABLEOLD : BOOL := FALSE;
END_VAR
END_FUNCTION_BLOCK

METHOD FB_RESET : BOOL
END_METHOD

(* ---- L_MC4P_READPARAMETER.pou ---- *)
FUNCTION_BLOCK L_MC4P_READPARAMETER EXTENDS L_MC4P_Template_AG_KIN
VAR_INPUT
	XENABLE : BOOL;
	DIPARAMETERNUMBER : DINT;
END_VAR
VAR_OUTPUT
	XVALID : BOOL;
	XBUSY : BOOL;
	XERROR : BOOL;
	EERRORID : L_IE1P_Error;
	LRVALUE : LREAL;
END_VAR
VAR
	XENABLEOLD : BOOL := FALSE;
END_VAR
END_FUNCTION_BLOCK

METHOD FB_RESET : BOOL
END_METHOD

(* ---- L_MC4P_SETACTIVETOOL.pou ---- *)
FUNCTION_BLOCK L_MC4P_SETACTIVETOOL EXTENDS L_MC4P_Template_AG_KIN
VAR_INPUT
	XEXECUTE : BOOL;
	ETOOLSYSTEM : L_MC4P_ToolSystem;
END_VAR
VAR_OUTPUT
	XDONE : BOOL;
	XBUSY : BOOL;
	XERROR : BOOL;
	EERRORID : L_IE1P_Error := L_IE1P_Error.NoError;
END_VAR
VAR
	XEXECUTEOLD : BOOL;
	XRESETOUTPUT : BOOL;
END_VAR
END_FUNCTION_BLOCK

(* ---- L_MC4P_SETTOOLTRANSFORM.pou ---- *)
FUNCTION_BLOCK L_MC4P_SETTOOLTRANSFORM EXTENDS L_MC4P_Template_AG_KIN
VAR_INPUT
	XEXECUTE : BOOL;
	SCTOOLPARAMETER : L_MC4P_TOOL_REF;
	ETOOLSYSTEM : L_MC4P_ToolSystem;
END_VAR
VAR_OUTPUT
	XDONE : BOOL;
	XBUSY : BOOL;
	XERROR : BOOL;
	EERRORID : L_IE1P_Error := L_IE1P_Error.NoError;
END_VAR
VAR
	PTOOL : POINTER TO L_MC4P_ToolTrafo;
	XEXECUTEOLD : BOOL;
	XRESETOUTPUT : BOOL;
	AXPARACCESSIBLE : ARRAY [1..7] OF BOOL;
	IDX : DINT;
	XINTERNALTESTMODE : BOOL := FALSE;
	INTERNALTESTMODE : BOOL;
END_VAR
END_FUNCTION_BLOCK

(* ---- L_MC4P_SETVALUEFILTER.pou ---- *)
FUNCTION_BLOCK L_MC4P_SETVALUEFILTER EXTENDS L_UBUP_MemoryProvider
VAR_INPUT
	XENABLE : BOOL;
	EFILTERMODE : L_MC4P_SetValueFilterMode := L_MC4P_SetValueFilterMode.EqualySpaced;
	UIFILTERTIME : UINT;
	LRSETPOSIN : LREAL;
	LRSETVELIN : LREAL;
	LRSETACCIN : LREAL;
	LRSETPOSINITIAL : LREAL;
	ETRAVERSINGRANGE : L_MC1P_TraversingRange := L_MC1P_TraversingRange.Limited;
	LRCYCLELENGTH : LREAL;
	LRINVCYCLELENGTH : LREAL;
END_VAR
VAR_OUTPUT
	XBUSY : BOOL;
	XACTIVE : BOOL;
	XERROR : BOOL;
	EERRORID : L_IE1P.L_IE1P_Error;
	DWINTERNALID : DWORD;
	LRSETPOSOUT : LREAL;
	LRSETVELOUT : LREAL;
	LRSETACCOUT : LREAL;
	LRACTFILTERDELAY : LREAL;
END_VAR
VAR
	LRTASKCYCLE : LREAL := -1;
	XENABLE_R : R_Trig;
	AMEM : ARRAY [1..4] OF ARRAY [1..cuiFilterSizeMax] OF LREAL;
	FB_AVG : L_USPP_AverageFilterRecursive;
	CUIFILTERSIZEMAX : UINT := 501;
	XRECURSIVE : BOOL := TRUE;
	PTR : POINTER TO BYTE;
	SIZE : UDINT;
END_VAR
END_FUNCTION_BLOCK

(* ---- L_MC4P_SIMPLETRANSFORMATION.pou ---- *)
FUNCTION_BLOCK L_MC4P_SIMPLETRANSFORMATION EXTENDS L_MC4P_TemplateTransformation
VAR
	SCSTORE : L_MC4P_IntermediateResultStore;
	SCSTORE_INTERNAL : L_MC4P_IntermediateResultStore;
END_VAR
END_FUNCTION_BLOCK

METHOD ADDTURNSTOJOINTS : L_IE1P_Error
VAR_INPUT
	PFLANGE_POS : POINTER TO ARRAY [1..6] OF LREAL;
	PJOINT_POS : POINTER TO ARRAY [1..6] OF LREAL;
END_VAR
VAR_IN_OUT
	SCTRAFOINFO : L_MC4P_TrafoInfo;
END_VAR
END_METHOD

METHOD CALCBACKWARDTRANSFORMATIONACC : L_IE1P_Error
VAR_INPUT
	PSTORE : POINTER TO L_MC4P_IntermediateResultStore;
END_VAR
VAR_IN_OUT
	SCTRAFOINFO : L_MC4P_TrafoInfo;
END_VAR
END_METHOD

METHOD CALCBACKWARDTRANSFORMATIONPOS : L_IE1P_Error
VAR_INPUT
	PSTORE : POINTER TO L_MC4P_IntermediateResultStore;
END_VAR
VAR_IN_OUT
	SCTRAFOINFO : L_MC4P_TrafoInfo;
END_VAR
END_METHOD

METHOD CALCBACKWARDTRANSFORMATIONVEL : L_IE1P_Error
VAR_INPUT
	PSTORE : POINTER TO L_MC4P_IntermediateResultStore;
END_VAR
VAR_IN_OUT
	SCTRAFOINFO : L_MC4P_TrafoInfo;
END_VAR
END_METHOD

METHOD CALCFORWARDTRANSFORMATIONACC : L_IE1P_Error
VAR_INPUT
	PSTORE : POINTER TO L_MC4P_IntermediateResultStore;
END_VAR
VAR_IN_OUT
	SCTRAFOINFO : L_MC4P_TrafoInfo;
END_VAR
END_METHOD

METHOD CALCFORWARDTRANSFORMATIONPOS : L_IE1P_Error
VAR_INPUT
	PSTORE : POINTER TO L_MC4P_IntermediateResultStore;
END_VAR
VAR_IN_OUT
	SCTRAFOINFO : L_MC4P_TrafoInfo;
END_VAR
END_METHOD

METHOD CALCFORWARDTRANSFORMATIONVEL : L_IE1P_Error
VAR_INPUT
	PSTORE : POINTER TO L_MC4P_IntermediateResultStore;
END_VAR
VAR_IN_OUT
	SCTRAFOINFO : L_MC4P_TrafoInfo;
END_VAR
END_METHOD

METHOD FB_INIT : BOOL
VAR_INPUT
	BINITRETAINS : BOOL;
	BINCOPYCODE : BOOL;
END_VAR
END_METHOD

METHOD CALCDINVERSEJACOBIAN : BOOL
VAR_INPUT
	ICOORDPROVIDER : L_MC4P_IKinCoordProvider;
	PDINVJACOBIAN : POINTER TO ARRAY [1..6, 1..6] OF LREAL;
END_VAR
VAR_OUTPUT
	SCERROR : L_MC4P_ErrorStruct;
END_VAR
END_METHOD

METHOD CALCDJACOBIAN : BOOL
VAR_INPUT
	ICOORDPROVIDER : L_MC4P_IKinCoordProvider;
	PDJACOBIAN : POINTER TO ARRAY [1..6, 1..6] OF LREAL;
END_VAR
VAR_OUTPUT
	SCERROR : L_MC4P_ErrorStruct;
END_VAR
END_METHOD

METHOD CALCINVERSEJACOBIAN : BOOL
VAR_INPUT
	ICOORDPROVIDER : L_MC4P_IKinCoordProvider;
	PINVJACOBIAN : POINTER TO ARRAY [1..6, 1..6] OF LREAL;
END_VAR
VAR_OUTPUT
	SCERROR : L_MC4P_ErrorStruct;
END_VAR
END_METHOD

METHOD CALCJACOBIAN : BOOL
VAR_INPUT
	ICOORDPROVIDER : L_MC4P_IKinCoordProvider;
	PJACOBIAN : POINTER TO ARRAY [1..6, 1..6] OF LREAL;
END_VAR
VAR_OUTPUT
	SCERROR : L_MC4P_ErrorStruct;
END_VAR
END_METHOD

METHOD MCS_ORIENTATIONCHECK : L_IE1P_Error
VAR_IN_OUT
	ICOORDPROVIDER : L_MC4P_KinCoordProvider;
END_VAR
END_METHOD

(* ---- L_MC4P_TCPFORCEOBSERVER.pou ---- *)
FUNCTION_BLOCK L_MC4P_TCPFORCEOBSERVER EXTENDS L_MC4P_Template_AG_KIN
VAR_INPUT
	XENABLE : BOOL;
	XUSEAXESGROUPPARAM : BOOL := FALSE;
	LRLOADMASS : LREAL;
	ITFDYNAMICPAR : L_MC4P_DynamicPar;
	LROBSERVATIONDYNAMIC : LREAL;
	EOBSERVATIONMODE : L_MC4P_ObservationMode;
END_VAR
VAR_OUTPUT
	XVALID : BOOL;
	XBUSY : BOOL;
	XERROR : BOOL;
	EERRORID : L_IE1P_Error;
	ALROBSERVEDTCPFORCE : ARRAY [1..3] OF LREAL;
	LROBSERVEDLOADMASS : LREAL;
END_VAR
VAR
	LICHANDLING : L_IMHP_LLMHandling;
	ALRGRAVITATION : ARRAY [1..3] OF LREAL;
	ALRCOULOMBFRIC : ARRAY [1..6] OF LREAL;
	ALRVISCFRIC : ARRAY [1..6] OF LREAL;
	ALRDYNAMICPAR : ARRAY [1..L_MC4P_Constants.uimaxNbrOfDynamicPar] OF LREAL;
	PLRREGRESSIONMATRIX : POINTER TO LREAL;
	XENABLEOLD : BOOL;
	EERRORTMP : L_IE1P_Error;
	ITFJACOBIAN : L_MC4P_IJacobi;
	ALRACTTORQUEACS : ARRAY [1..6] OF LREAL;
	ALRACTTORQUEJCS : ARRAY [1..6] OF LREAL;
	ALRCALCULATEDTORQUEJCS : ARRAY [1..6] OF LREAL;
	ALREXTTORQUE : ARRAY [1..6] OF LREAL;
	ALRTORQUEERROR : ARRAY [1..6] OF LREAL;
	ALRINVJACOBIAN : ARRAY [1..6, 1..6] OF LREAL;
	ALRTRANSPOSEDINVJACOBIAN : ARRAY [1..6, 1..6] OF LREAL;
	ALROBSERVEDTCPFORCEINT : ARRAY [1..6] OF LREAL;
	LROBSERVEDLOADMASSINT : LREAL;
	LROBSERVATIONDYNAMICLIM : LREAL;
	LROBSERVATIONDYNAMICINT : LREAL;
	APT1_ACTJCSPOS : ARRAY [1..6] OF L_USPP.L_USPP_PT1Filter;
	APT1_ACTJCSVEL : ARRAY [1..6] OF L_USPP.L_USPP_PT1Filter;
	APT1_ACTJCSACC : ARRAY [1..6] OF L_USPP.L_USPP_PT1Filter;
	APT1_ACTFCSPOS : ARRAY [1..6] OF L_USPP.L_USPP_PT1Filter;
	APT1_ACTFCSVEL : ARRAY [1..6] OF L_USPP.L_USPP_PT1Filter;
	APT1_ACTFCSACC : ARRAY [1..6] OF L_USPP.L_USPP_PT1Filter;
	APT1_ACTTORQUE : ARRAY [1..6] OF L_USPP.L_USPP_PT1Filter;
	AGOF : ARRAY [1..3] OF L_UMTP_GoodnessOfFit;
	LRCONVERGENCE : LREAL;
	LRVALIDTHRESHOLDON : LREAL := 0.75;
	LRVALIDTHRESHOLDOFF : LREAL := 0.5;
	RLS1 : L_UMTP_RLS;
	MASSMEANFILTER : L_MC4P_AvgValueFilter1D;
	AFORCEMEANFILTER : ARRAY [1..3] OF L_MC4P_AvgValueFilter1D;
	LRPT1FILTERTIME : LREAL;
	LRLAMBDA : LREAL;
	UIMEANFILTERTIME : UINT;
	XDIFFERENTIALDRIVE1ACTIVE : BOOL;
	PACTTRAFOEXTENSION1 : POINTER TO L_MC4P_TrafoExtensionBase;
	USINBROFDYNPAR : USINT;
	IDX : INT;
END_VAR
END_FUNCTION_BLOCK

METHOD CALCULATEMODEL
VAR_IN_OUT
	AXESGROUP : AXES_GROUP_KIN;
END_VAR
END_METHOD

(* ---- L_MC4P_TEACHCOORDINATESYSTEM.pou ---- *)
FUNCTION_BLOCK L_MC4P_TEACHCOORDINATESYSTEM EXTENDS L_MC4P_Template_AG_KIN
VAR_INPUT
	XEXECUTE : BOOL;
	XSTEPCONFIRM : BOOL;
	ECOORDSYSTEM : L_MC4P_CoordSystem;
END_VAR
VAR_OUTPUT
	XDONE : BOOL;
	XBUSY : BOOL;
	XERROR : BOOL;
	EERRORID : L_IE1P_Error;
	ENEXTSTEP : L_MC4P_TeachCoordinateSystemSteps;
	SCCOORDINATETRANSFORM : MC_COORD_REF;
END_VAR
VAR
	XEXECUTEOLD : BOOL;
	XSTEPCONFIRMOLD : BOOL;
	BASE_POS : ARRAY [1..3] OF LREAL;
	POS_TMP : ARRAY [1..3] OF LREAL;
	POS_TMP2 : ARRAY [1..3] OF LREAL;
	X_VEK : ARRAY [1..3] OF LREAL;
	Y_VEK : ARRAY [1..3] OF LREAL;
	Z_VEK : ARRAY [1..3] OF LREAL;
	XY_VEK : ARRAY [1..3] OF LREAL;
	T : ARRAY [1..4, 1..4] OF LREAL;
	MC_SETCOORDINATETRANSFORM1 : MC_SetCoordinateTransform;
END_VAR
END_FUNCTION_BLOCK

METHOD SETERROR
END_METHOD

(* ---- L_MC4P_TEMPLATE_AG_KIN.pou ---- *)
FUNCTION_BLOCK L_MC4P_TEMPLATE_AG_KIN EXTENDS L_MC4P_Template_ForAG
VAR_IN_OUT
	AXESGROUP : AXES_GROUP_KIN;
END_VAR
VAR
	SINSTANCESTR : STRING;
	AXESGROUP_WINITSTATEOLD : WORD;
END_VAR
END_FUNCTION_BLOCK

METHOD AXESGROUPINITDONE : BOOL
VAR_INPUT
	XEXECUTE : BOOL;
END_VAR
VAR_IN_OUT
	XERROR : BOOL;
	EERRORID : L_IE1P_Error;
	AXESGROUP : AXES_GROUP_KIN;
END_VAR
END_METHOD

METHOD FB_GETERRORITFID : DWORD
END_METHOD

METHOD FB_RESETERROR
VAR_INPUT
	XERROR : BOOL;
	WERRORID : WORD;
END_VAR
END_METHOD

METHOD FB_SETERROR
VAR_INPUT
	WERRORID : L_IE1P_Error := L_IE1P_Error.NoError;
	XSETERRORSTOP : BOOL := FALSE;
END_VAR
END_METHOD

METHOD FB_SETERRORINT
VAR_INPUT
	WERRORID : L_IE1P_Error := L_IE1P_Error.NoError;
	DWINTERNALID : DWORD;
	XSETERRORSTOP : BOOL := FALSE;
END_VAR
END_METHOD

METHOD FB_INIT : BOOL
VAR_INPUT
	BINITRETAINS : BOOL;
	BINCOPYCODE : BOOL;
END_VAR
END_METHOD

(* ---- L_MC4P_TEMPLATE_AG_KIN_LICENCE.pou ---- *)
FUNCTION_BLOCK L_MC4P_TEMPLATE_AG_KIN_LICENCE EXTENDS L_MC4P_Template_AG_KIN
VAR
	LICHANDLING : L_IMHP_LLMHandling;
	MC1P_LICENCE : L_MC1P_Template_Licence_150;
END_VAR
END_FUNCTION_BLOCK

METHOD ACTIVATEAPPCREDIT : BOOL
VAR_INPUT
	XACTIVATE : BOOL;
END_VAR
END_METHOD

(* ---- L_MC4P_TEMPLATE_AG_REF.pou ---- *)
FUNCTION_BLOCK L_MC4P_TEMPLATE_AG_REF EXTENDS L_MC4P_Template_ForAG
VAR_IN_OUT
	AXESGROUP : AXES_GROUP_REF;
END_VAR
VAR
	SINSTANCESTR : STRING;
	AXESGROUP_WINITSTATEOLD : WORD;
END_VAR
END_FUNCTION_BLOCK

METHOD AXESGROUPINITDONE : BOOL
VAR_INPUT
	XEXECUTE : BOOL;
END_VAR
VAR_IN_OUT
	XERROR : BOOL;
	EERRORID : L_IE1P_Error;
	AXESGROUP : AXES_GROUP_REF;
END_VAR
END_METHOD

METHOD FB_GETERRORITFID : DWORD
END_METHOD

METHOD FB_RESETERROR
VAR_INPUT
	XERROR : BOOL;
	WERRORID : WORD;
END_VAR
END_METHOD

METHOD FB_SETERROR
VAR_INPUT
	WERRORID : L_IE1P_Error := L_IE1P_Error.NoError;
	XSETERRORSTOP : BOOL := FALSE;
END_VAR
END_METHOD

METHOD FB_SETERRORINT
VAR_INPUT
	WERRORID : L_IE1P_Error := L_IE1P_Error.NoError;
	DWINTERNALID : DWORD;
	XSETERRORSTOP : BOOL := FALSE;
END_VAR
END_METHOD

METHOD FB_INIT : BOOL
VAR_INPUT
	BINITRETAINS : BOOL;
	BINCOPYCODE : BOOL;
END_VAR
END_METHOD
